PROPERTY PUBLIC Value : ETcVnKeypointDetectionTypeFAST
GET
Value := activeData;
END_GET
SET
activeData := Value;
END_SET
END_PROPERTY

END_FUNCTION_BLOCK

// Datatypes/Enums/_ETcVnLineType
{attribute 'linkalways'} 
{attribute 'no_explicit_call' := 'This FB is a CLASS and must be accessed using methods or properties'}
{attribute 'enable_dynamic_creation'}
FUNCTION_BLOCK _ETcVnLineType EXTENDS EnumDatatypeBase
VAR
	localData : ETcVnLineType;
	activeData : REFERENCE TO ETcVnLineType;
	enumBaseDatatype : _DINT(localData);
END_VAR

METHOD PROTECTED SetBaseDatatypeReference
VAR_INPUT
END_VAR
enumBaseDatatype.MakeReferenceTo(activeData);
END_METHOD

PROPERTY PUBLIC Address : PVOID
GET
Address := ADR(activeData);
END_GET
END_PROPERTY

METHOD PUBLIC ClearReference
VAR_INPUT
END_VAR
activeData REF= localData;
SetBaseDatatypeReference();
END_METHOD

PROPERTY PUBLIC Size : UDINT
GET
Size := SIZEOF(activeData);
END_GET
END_PROPERTY

METHOD FB_init : BOOL
VAR_INPUT
	bInitRetains : BOOL; // if TRUE, the retain variables are initialized (warm start / cold start)
	bInCopyCode : BOOL;  // if TRUE, the instance afterwards gets moved into the copy code (online change)
	InitialValue : ETcVnLineType;
END_VAR
localData := InitialValue;
AddBaseDatatype(enumBaseDatatype);
ClearReference();

AddLocalEnumeration('TCVN_LT_4_CONNECTED', ETcVnLineType.TCVN_LT_4_CONNECTED);
AddLocalEnumeration('TCVN_LT_8_CONNECTED', ETcVnLineType.TCVN_LT_8_CONNECTED);
AddLocalEnumeration('TCVN_LT_ANTIALIASED', ETcVnLineType.TCVN_LT_ANTIALIASED);
END_METHOD

METHOD PRIVATE AddLocalEnumeration
VAR_INPUT
	Enumeration : T_MAXSTRING;
	Value : ETcVnLineType;
END_VAR
AddEnumeration(Enumeration, Value);
END_METHOD

METHOD IsEnumeratorValueEqual : BOOL
VAR_INPUT
	Enumerator : I_KeyValueForwardEnumerator;
END_VAR
VAR
	storedValue : ETcVnLineType;
END_VAR
IF NOT Enumerator.TryGet(storedValue) THEN
	RETURN;
END_IF

IsEnumeratorValueEqual := storedValue = activeData;
END_METHOD

METHOD PUBLIC Clone : I_Datatype
VAR
    pClone : POINTER TO _ETcVnLineType;
END_VAR
pClone := __NEW(_ETcVnLineType(InitialValue := Value));
Clone := pClone^;
END_METHOD

PROPERTY PUBLIC Identifier : T_MAXSTRING
GET
Identifier := 'ETcVnLineType';
END_GET
END_PROPERTY

METHOD PUBLIC MakeReferenceTo
VAR_INPUT
	ReferenceTarget : REFERENCE TO ETcVnLineType;
END_VAR
activeData REF= ReferenceTarget;
SetBaseDatatypeReference();
END_METHOD

METHOD TryMakeReferenceTo : BOOL
VAR_INPUT
	Target : I_Datatype;
END_VAR
VAR
	pTargetData : POINTER TO ETcVnLineType;
END_VAR
IF NOT IsEquivalentTo(Target) THEN
	RETURN;
END_IF

pTargetData := Target.Address;
activeData REF= pTargetData^;
SetBaseDatatypeReference();
TryMakeReferenceTo := TRUE;
END_METHOD

PROPERTY PUBLIC Value : ETcVnLineType
GET
Value := activeData;
END_GET
SET
activeData := Value;
END_SET
END_PROPERTY

END_FUNCTION_BLOCK

// Datatypes/Enums/_ETcVnMorphologicalOperator
{attribute 'linkalways'} 
{attribute 'no_explicit_call' := 'This FB is a CLASS and must be accessed using methods or properties'}
{attribute 'enable_dynamic_creation'}
FUNCTION_BLOCK _ETcVnMorphologicalOperator EXTENDS EnumDatatypeBase
VAR
	localData : ETcVnMorphologicalOperator;
	activeData : REFERENCE TO ETcVnMorphologicalOperator;
	enumBaseDatatype : _DINT(localData);
END_VAR

METHOD PROTECTED SetBaseDatatypeReference
VAR_INPUT
END_VAR
enumBaseDatatype.MakeReferenceTo(activeData);
END_METHOD

PROPERTY PUBLIC Address : PVOID
GET
Address := ADR(activeData);
END_GET
END_PROPERTY

METHOD PUBLIC ClearReference
VAR_INPUT
END_VAR
activeData REF= localData;
SetBaseDatatypeReference();
END_METHOD

PROPERTY PUBLIC Size : UDINT
GET
Size := SIZEOF(activeData);
END_GET
END_PROPERTY

METHOD FB_init : BOOL
VAR_INPUT
	bInitRetains : BOOL; // if TRUE, the retain variables are initialized (warm start / cold start)
	bInCopyCode : BOOL;  // if TRUE, the instance afterwards gets moved into the copy code (online change)
	InitialValue : ETcVnMorphologicalOperator;
END_VAR
localData := InitialValue;
AddBaseDatatype(enumBaseDatatype);
ClearReference();

AddLocalEnumeration('TCVN_MO_EROSION', ETcVnMorphologicalOperator.TCVN_MO_EROSION);
AddLocalEnumeration('TCVN_MO_DILATION', ETcVnMorphologicalOperator.TCVN_MO_DILATION);
AddLocalEnumeration('TCVN_MO_OPENING', ETcVnMorphologicalOperator.TCVN_MO_OPENING);
AddLocalEnumeration('TCVN_MO_CLOSING', ETcVnMorphologicalOperator.TCVN_MO_CLOSING);
AddLocalEnumeration('TCVN_MO_GRADIENT', ETcVnMorphologicalOperator.TCVN_MO_GRADIENT);
AddLocalEnumeration('TCVN_MO_WHITE_TOPHAT', .TCVN_MO_WHITE_TOPHAT);
AddLocalEnumeration('TCVN_MO_BLACK_TOPHAT', ETcVnMorphologicalOperator.TCVN_MO_BLACK_TOPHAT);
AddLocalEnumeration('TCVN_MO_OPENING_BY_RECONSTRUCTION', ETcVnMorphologicalOperator.TCVN_MO_OPENING_BY_RECONSTRUCTION);
AddLocalEnumeration('TCVN_MO_CLOSING_BY_RECONSTRUCTION', ETcVnMorphologicalOperator.TCVN_MO_CLOSING_BY_RECONSTRUCTION);
AddLocalEnumeration('TCVN_MO_WHITE_TOPHAT_BY_RECONSTRUCTION', ETcVnMorphologicalOperator.TCVN_MO_WHITE_TOPHAT_BY_RECONSTRUCTION);
AddLocalEnumeration('TCVN_MO_BLACK_TOPHAT_BY_RECONSTRUCTION', ETcVnMorphologicalOperator.TCVN_MO_BLACK_TOPHAT_BY_RECONSTRUCTION);
END_METHOD

METHOD PRIVATE AddLocalEnumeration
VAR_INPUT
	Enumeration : T_MAXSTRING;
	Value : ETcVnMorphologicalOperator;
END_VAR
AddEnumeration(Enumeration, Value);
END_METHOD

METHOD IsEnumeratorValueEqual : BOOL
VAR_INPUT
	Enumerator : I_KeyValueForwardEnumerator;
END_VAR
VAR
	storedValue : ETcVnMorphologicalOperator;
END_VAR
IF NOT Enumerator.TryGet(storedValue) THEN
	RETURN;
END_IF

IsEnumeratorValueEqual := storedValue = activeData;
END_METHOD

METHOD PUBLIC Clone : I_Datatype
VAR
    pClone : POINTER TO _ETcVnMorphologicalOperator;
END_VAR
pClone := __NEW(_ETcVnMorphologicalOperator(InitialValue := Value));
Clone := pClone^;
END_METHOD

PROPERTY PUBLIC Identifier : T_MAXSTRING
GET
Identifier := 'ETcVnMorphologicalOperator';
END_GET
END_PROPERTY

METHOD PUBLIC MakeReferenceTo
VAR_INPUT
	ReferenceTarget : REFERENCE TO ETcVnMorphologicalOperator;
END_VAR
activeData REF= ReferenceTarget;
SetBaseDatatypeReference();
END_METHOD

METHOD TryMakeReferenceTo : BOOL
VAR_INPUT
	Target : I_Datatype;
END_VAR
VAR
	pTargetData : POINTER TO ETcVnMorphologicalOperator;
END_VAR
IF NOT IsEquivalentTo(Target) THEN
	RETURN;
END_IF

pTargetData := Target.Address;
activeData REF= pTargetData^;
SetBaseDatatypeReference();
TryMakeReferenceTo := TRUE;
END_METHOD

PROPERTY PUBLIC Value : ETcVnMorphologicalOperator
GET
Value := activeData;
END_GET
SET
activeData := Value;
END_SET
END_PROPERTY

END_FUNCTION_BLOCK

// Datatypes/Enums/_ETcVnNormalizationType
{attribute 'linkalways'} 
{attribute 'no_explicit_call' := 'This FB is a CLASS and must be accessed using methods or properties'}
{attribute 'enable_dynamic_creation'}
FUNCTION_BLOCK _ETcVnNormalizationType EXTENDS EnumDatatypeBase
VAR
	localData : ETcVnNormalizationType;
	activeData : REFERENCE TO ETcVnNormalizationType;
	enumBaseDatatype : _DINT(localData);
END_VAR

METHOD PROTECTED SetBaseDatatypeReference
VAR_INPUT
END_VAR
enumBaseDatatype.MakeReferenceTo(activeData);
END_METHOD

PROPERTY PUBLIC Address : PVOID
GET
Address := ADR(activeData);
END_GET
END_PROPERTY

METHOD PUBLIC ClearReference
VAR_INPUT
END_VAR
activeData REF= localData;
SetBaseDatatypeReference();
END_METHOD

PROPERTY PUBLIC Size : UDINT
GET
Size := SIZEOF(activeData);
END_GET
END_PROPERTY

METHOD FB_init : BOOL
VAR_INPUT
	bInitRetains : BOOL; // if TRUE, the retain variables are initialized (warm start / cold start)
	bInCopyCode : BOOL;  // if TRUE, the instance afterwards gets moved into the copy code (online change)
	InitialValue : ETcVnNormalizationType;
END_VAR
localData := InitialValue;
AddBaseDatatype(enumBaseDatatype);
ClearReference();

AddLocalEnumeration('TCVN_NT_INF', ETcVnNormalizationType.TCVN_NT_INF);
AddLocalEnumeration('TCVN_NT_L1', ETcVnNormalizationType.TCVN_NT_L1);
AddLocalEnumeration('TCVN_NT_L2', ETcVnNormalizationType.TCVN_NT_L2);
AddLocalEnumeration('TCVN_NT_L2SQR', ETcVnNormalizationType.TCVN_NT_L2SQR);
AddLocalEnumeration('TCVN_NT_HAMMING', ETcVnNormalizationType.TCVN_NT_HAMMING);
AddLocalEnumeration('TCVN_NT_HAMMING2', ETcVnNormalizationType.TCVN_NT_HAMMING2);
AddLocalEnumeration('TCVN_NT_RELATIVE_INF', ETcVnNormalizationType.TCVN_NT_RELATIVE_INF);
AddLocalEnumeration('TCVN_NT_RELATIVE_L1', ETcVnNormalizationType.TCVN_NT_RELATIVE_L1);
AddLocalEnumeration('TCVN_NT_RELATIVE_L2', ETcVnNormalizationType.TCVN_NT_RELATIVE_L2);
AddLocalEnumeration('TCVN_NT_RELATIVE_L2SQR', ETcVnNormalizationType.TCVN_NT_RELATIVE_L2SQR);
AddLocalEnumeration('TCVN_NT_RELATIVE_HAMMING', ETcVnNormalizationType.TCVN_NT_RELATIVE_HAMMING);
AddLocalEnumeration('TCVN_NT_RELATIVE_HAMMING2', ETcVnNormalizationType.TCVN_NT_RELATIVE_HAMMING2);
AddLocalEnumeration('TCVN_NT_MINMAX', ETcVnNormalizationType.TCVN_NT_MINMAX);
END_METHOD

METHOD PRIVATE AddLocalEnumeration
VAR_INPUT
	Enumeration : T_MAXSTRING;
	Value : ETcVnNormalizationType;
END_VAR
AddEnumeration(Enumeration, Value);
END_METHOD

METHOD IsEnumeratorValueEqual : BOOL
VAR_INPUT
	Enumerator : I_KeyValueForwardEnumerator;
END_VAR
VAR
	storedValue : ETcVnNormalizationType;
END_VAR
IF NOT Enumerator.TryGet(storedValue) THEN
	RETURN;
END_IF

IsEnumeratorValueEqual := storedValue = activeData;
END_METHOD

METHOD PUBLIC Clone : I_Datatype
VAR
    pClone : POINTER TO _ETcVnNormalizationType;
END_VAR
pClone := __NEW(_ETcVnNormalizationType(InitialValue := Value));
Clone := pClone^;
END_METHOD

PROPERTY PUBLIC Identifier : T_MAXSTRING
GET
Identifier := 'ETcVnNormalizationType';
END_GET
END_PROPERTY

METHOD PUBLIC MakeReferenceTo
VAR_INPUT
	ReferenceTarget : REFERENCE TO ETcVnNormalizationType;
END_VAR
activeData REF= ReferenceTarget;
SetBaseDatatypeReference();
END_METHOD

METHOD TryMakeReferenceTo : BOOL
VAR_INPUT
	Target : I_Datatype;
END_VAR
VAR
	pTargetData : POINTER TO ETcVnNormalizationType;
END_VAR
IF NOT IsEquivalentTo(Target) THEN
	RETURN;
END_IF

pTargetData := Target.Address;
activeData REF= pTargetData^;
SetBaseDatatypeReference();
TryMakeReferenceTo := TRUE;
END_METHOD

PROPERTY PUBLIC Value : ETcVnNormalizationType
GET
Value := activeData;
END_GET
SET
activeData := Value;
END_SET
END_PROPERTY

END_FUNCTION_BLOCK

// Datatypes/Enums/_ETcVnOrientationMethod
{attribute 'linkalways'} 
{attribute 'no_explicit_call' := 'This FB is a CLASS and must be accessed using methods or properties'}
{attribute 'enable_dynamic_creation'}
FUNCTION_BLOCK _ETcVnOrientationMethod EXTENDS EnumDatatypeBase
VAR
	localData : ETcVnOrientationMethod;
	activeData : REFERENCE TO ETcVnOrientationMethod;
	enumBaseDatatype : _DINT(localData);
END_VAR

METHOD PROTECTED SetBaseDatatypeReference
VAR_INPUT
END_VAR
enumBaseDatatype.MakeReferenceTo(activeData);
END_METHOD

PROPERTY PUBLIC Address : PVOID
GET
Address := ADR(activeData);
END_GET
END_PROPERTY

METHOD PUBLIC ClearReference
VAR_INPUT
END_VAR
activeData REF= localData;
SetBaseDatatypeReference();
END_METHOD

PROPERTY PUBLIC Size : UDINT
GET
Size := SIZEOF(activeData);
END_GET
END_PROPERTY

METHOD FB_init : BOOL
VAR_INPUT
	bInitRetains : BOOL; // if TRUE, the retain variables are initialized (warm start / cold start)
	bInCopyCode : BOOL;  // if TRUE, the instance afterwards gets moved into the copy code (online change)
	InitialValue : ETcVnOrientationMethod;
END_VAR
localData := InitialValue;
AddBaseDatatype(enumBaseDatatype);
ClearReference();

AddLocalEnumeration('TCVN_OM_PCA', ETcVnOrientationMethod.TCVN_OM_PCA);
AddLocalEnumeration('TCVN_OM_FITELLIPSE', ETcVnOrientationMethod.TCVN_OM_FITELLIPSE);
AddLocalEnumeration('TCVN_OM_MOMENTS', ETcVnOrientationMethod.TCVN_OM_MOMENTS);
AddLocalEnumeration('TCVN_OM_ENCLOSINGRECT', ETcVnOrientationMethod.TCVN_OM_ENCLOSINGRECT);
END_METHOD

METHOD PRIVATE AddLocalEnumeration
VAR_INPUT
	Enumeration : T_MAXSTRING;
	Value : ETcVnOrientationMethod;
END_VAR
AddEnumeration(Enumeration, Value);
END_METHOD

METHOD IsEnumeratorValueEqual : BOOL
VAR_INPUT
	Enumerator : I_KeyValueForwardEnumerator;
END_VAR
VAR
	storedValue : ETcVnOrientationMethod;
END_VAR
IF NOT Enumerator.TryGet(storedValue) THEN
	RETURN;
END_IF

IsEnumeratorValueEqual := storedValue = activeData;
END_METHOD

METHOD PUBLIC Clone : I_Datatype
VAR
    pClone : POINTER TO _ETcVnOrientationMethod;
END_VAR
pClone := __NEW(_ETcVnOrientationMethod(InitialValue := Value));
Clone := pClone^;
END_METHOD

PROPERTY PUBLIC Identifier : T_MAXSTRING
GET
Identifier := 'ETcVnOrientationMethod';
END_GET
END_PROPERTY

METHOD PUBLIC MakeReferenceTo
VAR_INPUT
	ReferenceTarget : REFERENCE TO ETcVnOrientationMethod;
END_VAR
activeData REF= ReferenceTarget;
SetBaseDatatypeReference();
END_METHOD

METHOD TryMakeReferenceTo : BOOL
VAR_INPUT
	Target : I_Datatype;
END_VAR
VAR
	pTargetData : POINTER TO ETcVnOrientationMethod;
END_VAR
IF NOT IsEquivalentTo(Target) THEN
	RETURN;
END_IF

pTargetData := Target.Address;
activeData REF= pTargetData^;
SetBaseDatatypeReference();
TryMakeReferenceTo := TRUE;
END_METHOD

PROPERTY PUBLIC Value : ETcVnOrientationMethod
GET
Value := activeData;
END_GET
SET
activeData := Value;
END_SET
END_PROPERTY

END_FUNCTION_BLOCK

// Datatypes/Enums/_ETcVnPixelConnectivity
{attribute 'linkalways'} 
{attribute 'no_explicit_call' := 'This FB is a CLASS and must be accessed using methods or properties'}
{attribute 'enable_dynamic_creation'}
FUNCTION_BLOCK _ETcVnPixelConnectivity EXTENDS EnumDatatypeBase
VAR
	localData : ETcVnPixelConnectivity;
	activeData : REFERENCE TO ETcVnPixelConnectivity;
	enumBaseDatatype : _DINT(localData);
END_VAR

METHOD PROTECTED SetBaseDatatypeReference
VAR_INPUT
END_VAR
enumBaseDatatype.MakeReferenceTo(activeData);
END_METHOD

PROPERTY PUBLIC Address : PVOID
GET
Address := ADR(activeData);
END_GET
END_PROPERTY

METHOD PUBLIC ClearReference
VAR_INPUT
END_VAR
activeData REF= localData;
SetBaseDatatypeReference();
END_METHOD

PROPERTY PUBLIC Size : UDINT
GET
Size := SIZEOF(activeData);
END_GET
END_PROPERTY

METHOD FB_init : BOOL
VAR_INPUT
	bInitRetains : BOOL; // if TRUE, the retain variables are initialized (warm start / cold start)
	bInCopyCode : BOOL;  // if TRUE, the instance afterwards gets moved into the copy code (online change)
	InitialValue : ETcVnPixelConnectivity;
END_VAR
localData := InitialValue;
AddBaseDatatype(enumBaseDatatype);
ClearReference();

AddLocalEnumeration('TCVN_PC_4', ETcVnPixelConnectivity.TCVN_PC_4);
AddLocalEnumeration('TCVN_PC_8', ETcVnPixelConnectivity.TCVN_PC_8);
END_METHOD

METHOD PRIVATE AddLocalEnumeration
VAR_INPUT
	Enumeration : T_MAXSTRING;
	Value : ETcVnPixelConnectivity;
END_VAR
AddEnumeration(Enumeration, Value);
END_METHOD

METHOD IsEnumeratorValueEqual : BOOL
VAR_INPUT
	Enumerator : I_KeyValueForwardEnumerator;
END_VAR
VAR
	storedValue : ETcVnPixelConnectivity;
END_VAR
IF NOT Enumerator.TryGet(storedValue) THEN
	RETURN;
END_IF

IsEnumeratorValueEqual := storedValue = activeData;
END_METHOD

METHOD PUBLIC Clone : I_Datatype
VAR
    pClone : POINTER TO _ETcVnPixelConnectivity;
END_VAR
pClone := __NEW(_ETcVnPixelConnectivity(InitialValue := Value));
Clone := pClone^;
END_METHOD

PROPERTY PUBLIC Identifier : T_MAXSTRING
GET
Identifier := 'ETcVnPixelConnectivity';
END_GET
END_PROPERTY

METHOD PUBLIC MakeReferenceTo
VAR_INPUT
	ReferenceTarget : REFERENCE TO ETcVnPixelConnectivity;
END_VAR
activeData REF= ReferenceTarget;
SetBaseDatatypeReference();
END_METHOD

METHOD TryMakeReferenceTo : BOOL
VAR_INPUT
	Target : I_Datatype;
END_VAR
VAR
	pTargetData : POINTER TO ETcVnPixelConnectivity;
END_VAR
IF NOT IsEquivalentTo(Target) THEN
	RETURN;
END_IF

pTargetData := Target.Address;
activeData REF= pTargetData^;
SetBaseDatatypeReference();
TryMakeReferenceTo := TRUE;
END_METHOD

PROPERTY PUBLIC Value : ETcVnPixelConnectivity
GET
Value := activeData;
END_GET
SET
activeData := Value;
END_SET
END_PROPERTY

END_FUNCTION_BLOCK

// Datatypes/Enums/_ETcVnRectangleIntersection
{attribute 'linkalways'} 
{attribute 'no_explicit_call' := 'This FB is a CLASS and must be accessed using methods or properties'}
{attribute 'enable_dynamic_creation'}
FUNCTION_BLOCK _ETcVnRectangleIntersection EXTENDS EnumDatatypeBase
VAR
	localData : ETcVnRectangleIntersection;
	activeData : REFERENCE TO ETcVnRectangleIntersection;
	enumBaseDatatype : _DINT(localData);
END_VAR

METHOD PROTECTED SetBaseDatatypeReference
VAR_INPUT
END_VAR
enumBaseDatatype.MakeReferenceTo(activeData);
END_METHOD

PROPERTY PUBLIC Address : PVOID
GET
Address := ADR(activeData);
END_GET
END_PROPERTY

METHOD PUBLIC ClearReference
VAR_INPUT
END_VAR
activeData REF= localData;
SetBaseDatatypeReference();
END_METHOD

PROPERTY PUBLIC Size : UDINT
GET
Size := SIZEOF(activeData);
END_GET
END_PROPERTY

METHOD FB_init : BOOL
VAR_INPUT
	bInitRetains : BOOL; // if TRUE, the retain variables are initialized (warm start / cold start)
	bInCopyCode : BOOL;  // if TRUE, the instance afterwards gets moved into the copy code (online change)
	InitialValue : ETcVnRectangleIntersection;
END_VAR
localData := InitialValue;
AddBaseDatatype(enumBaseDatatype);
ClearReference();

AddLocalEnumeration('TCVN_RI_NONE', ETcVnRectangleIntersection.TCVN_RI_NONE);
AddLocalEnumeration('TCVN_RI_PARTIAL', ETcVnRectangleIntersection.TCVN_RI_PARTIAL);
AddLocalEnumeration('TCVN_RI_FULL', ETcVnRectangleIntersection.TCVN_RI_FULL);
END_METHOD

METHOD PRIVATE AddLocalEnumeration
VAR_INPUT
	Enumeration : T_MAXSTRING;
	Value : ETcVnRectangleIntersection;
END_VAR
AddEnumeration(Enumeration, Value);
END_METHOD

METHOD IsEnumeratorValueEqual : BOOL
VAR_INPUT
	Enumerator : I_KeyValueForwardEnumerator;
END_VAR
VAR
	storedValue : ETcVnRectangleIntersection;
END_VAR
IF NOT Enumerator.TryGet(storedValue) THEN
	RETURN;
END_IF

IsEnumeratorValueEqual := storedValue = activeData;
END_METHOD

METHOD PUBLIC Clone : I_Datatype
VAR
    pClone : POINTER TO _ETcVnRectangleIntersection;
END_VAR
pClone := __NEW(_ETcVnRectangleIntersection(InitialValue := Value));
Clone := pClone^;
END_METHOD

PROPERTY PUBLIC Identifier : T_MAXSTRING
GET
Identifier := 'ETcVnRectangleIntersection';
END_GET
END_PROPERTY

METHOD PUBLIC MakeReferenceTo
VAR_INPUT
	ReferenceTarget : REFERENCE TO ETcVnRectangleIntersection;
END_VAR
activeData REF= ReferenceTarget;
SetBaseDatatypeReference();
END_METHOD

METHOD TryMakeReferenceTo : BOOL
VAR_INPUT
	Target : I_Datatype;
END_VAR
VAR
	pTargetData : POINTER TO ETcVnRectangleIntersection;
END_VAR
IF NOT IsEquivalentTo(Target) THEN
	RETURN;
END_IF

pTargetData := Target.Address;
activeData REF= pTargetData^;
SetBaseDatatypeReference();
TryMakeReferenceTo := TRUE;
END_METHOD

PROPERTY PUBLIC Value : ETcVnRectangleIntersection
GET
Value := activeData;
END_GET
SET
activeData := Value;
END_SET
END_PROPERTY

END_FUNCTION_BLOCK

// Datatypes/Enums/_ETcVnRotationAngle
{attribute 'linkalways'} 
{attribute 'no_explicit_call' := 'This FB is a CLASS and must be accessed using methods or properties'}
{attribute 'enable_dynamic_creation'}
FUNCTION_BLOCK _ETcVnRotationAngle EXTENDS EnumDatatypeBase
VAR
	localData : ETcVnRotationAngle;
	activeData : REFERENCE TO ETcVnRotationAngle;
	enumBaseDatatype : _DINT(localData);
END_VAR

METHOD PROTECTED SetBaseDatatypeReference
VAR_INPUT
END_VAR
enumBaseDatatype.MakeReferenceTo(activeData);
END_METHOD

PROPERTY PUBLIC Address : PVOID
GET
Address := ADR(activeData);
END_GET
END_PROPERTY

METHOD PUBLIC ClearReference
VAR_INPUT
END_VAR
activeData REF= localData;
SetBaseDatatypeReference();
END_METHOD

PROPERTY PUBLIC Size : UDINT
GET
Size := SIZEOF(activeData);
END_GET
END_PROPERTY

METHOD FB_init : BOOL
VAR_INPUT
	bInitRetains : BOOL; // if TRUE, the retain variables are initialized (warm start / cold start)
	bInCopyCode : BOOL;  // if TRUE, the instance afterwards gets moved into the copy code (online change)
	InitialValue : ETcVnRotationAngle;
END_VAR
localData := InitialValue;
AddBaseDatatype(enumBaseDatatype);
ClearReference();

AddLocalEnumeration('TCVN_RA_90_DEG', ETcVnRotationAngle.TCVN_RA_90_DEG);
AddLocalEnumeration('TCVN_RA_180_DEG', ETcVnRotationAngle.TCVN_RA_180_DEG);
AddLocalEnumeration('TCVN_RA_270_DEG', ETcVnRotationAngle.TCVN_RA_270_DEG);
END_METHOD

METHOD PRIVATE AddLocalEnumeration
VAR_INPUT
	Enumeration : T_MAXSTRING;
	Value : ETcVnRotationAngle;
END_VAR
AddEnumeration(Enumeration, Value);
END_METHOD

METHOD IsEnumeratorValueEqual : BOOL
VAR_INPUT
	Enumerator : I_KeyValueForwardEnumerator;
END_VAR
VAR
	storedValue : ETcVnRotationAngle;
END_VAR
IF NOT Enumerator.TryGet(storedValue) THEN
	RETURN;
END_IF

IsEnumeratorValueEqual := storedValue = activeData;
END_METHOD

METHOD PUBLIC Clone : I_Datatype
VAR
    pClone : POINTER TO _ETcVnRotationAngle;
END_VAR
pClone := __NEW(_ETcVnRotationAngle(InitialValue := Value));
Clone := pClone^;
END_METHOD

PROPERTY PUBLIC Identifier : T_MAXSTRING
GET
Identifier := 'ETcVnRotationAngle';
END_GET
END_PROPERTY

METHOD PUBLIC MakeReferenceTo
VAR_INPUT
	ReferenceTarget : REFERENCE TO ETcVnRotationAngle;
END_VAR
activeData REF= ReferenceTarget;
SetBaseDatatypeReference();
END_METHOD

METHOD TryMakeReferenceTo : BOOL
VAR_INPUT
	Target : I_Datatype;
END_VAR
VAR
	pTargetData : POINTER TO ETcVnRotationAngle;
END_VAR
IF NOT IsEquivalentTo(Target) THEN
	RETURN;
END_IF

pTargetData := Target.Address;
activeData REF= pTargetData^;
SetBaseDatatypeReference();
TryMakeReferenceTo := TRUE;
END_METHOD

PROPERTY PUBLIC Value : ETcVnRotationAngle
GET
Value := activeData;
END_GET
SET
activeData := Value;
END_SET
END_PROPERTY

END_FUNCTION_BLOCK

// Datatypes/Enums/_ETcVnSignedNormalization
{attribute 'linkalways'} 
{attribute 'no_explicit_call' := 'This FB is a CLASS and must be accessed using methods or properties'}
{attribute 'enable_dynamic_creation'}
FUNCTION_BLOCK _ETcVnSignedNormalization EXTENDS EnumDatatypeBase
VAR
	localData : ETcVnSignedNormalization;
	activeData : REFERENCE TO ETcVnSignedNormalization;
	enumBaseDatatype : _INT(localData);
END_VAR

METHOD PROTECTED SetBaseDatatypeReference
VAR_INPUT
END_VAR
enumBaseDatatype.MakeReferenceTo(activeData);
END_METHOD

PROPERTY PUBLIC Address : PVOID
GET
Address := ADR(activeData);
END_GET
END_PROPERTY

METHOD PUBLIC ClearReference
VAR_INPUT
END_VAR
activeData REF= localData;
SetBaseDatatypeReference();
END_METHOD

PROPERTY PUBLIC Size : UDINT
GET
Size := SIZEOF(activeData);
END_GET
END_PROPERTY

METHOD FB_init : BOOL
VAR_INPUT
	bInitRetains : BOOL; // if TRUE, the retain variables are initialized (warm start / cold start)
	bInCopyCode : BOOL;  // if TRUE, the instance afterwards gets moved into the copy code (online change)
	InitialValue : ETcVnSignedNormalization;
END_VAR
localData := InitialValue;
AddBaseDatatype(enumBaseDatatype);
ClearReference();

AddLocalEnumeration('TCVN_SN_FIX_ZERO', ETcVnSignedNormalization.TCVN_SN_FIX_ZERO);
AddLocalEnumeration('TCVN_SN_FULL_SCALE', ETcVnSignedNormalization.TCVN_SN_FULL_SCALE);
END_METHOD

METHOD PRIVATE AddLocalEnumeration
VAR_INPUT
	Enumeration : T_MAXSTRING;
	Value : ETcVnSignedNormalization;
END_VAR
AddEnumeration(Enumeration, Value);
END_METHOD

METHOD IsEnumeratorValueEqual : BOOL
VAR_INPUT
	Enumerator : I_KeyValueForwardEnumerator;
END_VAR
VAR
	storedValue : ETcVnSignedNormalization;
END_VAR
IF NOT Enumerator.TryGet(storedValue) THEN
	RETURN;
END_IF

IsEnumeratorValueEqual := storedValue = activeData;
END_METHOD

METHOD PUBLIC Clone : I_Datatype
VAR
    pClone : POINTER TO _ETcVnSignedNormalization;
END_VAR
pClone := __NEW(_ETcVnSignedNormalization(InitialValue := Value));
Clone := pClone^;
END_METHOD

PROPERTY PUBLIC Identifier : T_MAXSTRING
GET
Identifier := 'ETcVnSignedNormalization';
END_GET
END_PROPERTY

METHOD PUBLIC MakeReferenceTo
VAR_INPUT
	ReferenceTarget : REFERENCE TO ETcVnSignedNormalization;
END_VAR
activeData REF= ReferenceTarget;
SetBaseDatatypeReference();
END_METHOD

METHOD TryMakeReferenceTo : BOOL
VAR_INPUT
	Target : I_Datatype;
END_VAR
VAR
	pTargetData : POINTER TO ETcVnSignedNormalization;
END_VAR
IF NOT IsEquivalentTo(Target) THEN
	RETURN;
END_IF

pTargetData := Target.Address;
activeData REF= pTargetData^;
SetBaseDatatypeReference();
TryMakeReferenceTo := TRUE;
END_METHOD

PROPERTY PUBLIC Value : ETcVnSignedNormalization
GET
Value := activeData;
END_GET
SET
activeData := Value;
END_SET
END_PROPERTY

END_FUNCTION_BLOCK

// Datatypes/Enums/_ETcVnStructuringElementShape
{attribute 'linkalways'} 
{attribute 'no_explicit_call' := 'This FB is a CLASS and must be accessed using methods or properties'}
{attribute 'enable_dynamic_creation'}
FUNCTION_BLOCK _ETcVnStructuringElementShape EXTENDS EnumDatatypeBase
VAR
	localData : ETcVnStructuringElementShape;
	activeData : REFERENCE TO ETcVnStructuringElementShape;
	enumBaseDatatype : _DINT(localData);
END_VAR

METHOD PROTECTED SetBaseDatatypeReference
VAR_INPUT
END_VAR
enumBaseDatatype.MakeReferenceTo(activeData);
END_METHOD

PROPERTY PUBLIC Address : PVOID
GET
Address := ADR(activeData);
END_GET
END_PROPERTY

METHOD PUBLIC ClearReference
VAR_INPUT
END_VAR
activeData REF= localData;
SetBaseDatatypeReference();
END_METHOD

PROPERTY PUBLIC Size : UDINT
GET
Size := SIZEOF(activeData);
END_GET
END_PROPERTY

METHOD FB_init : BOOL
VAR_INPUT
	bInitRetains : BOOL; // if TRUE, the retain variables are initialized (warm start / cold start)
	bInCopyCode : BOOL;  // if TRUE, the instance afterwards gets moved into the copy code (online change)
	InitialValue : ETcVnStructuringElementShape;
END_VAR
localData := InitialValue;
AddBaseDatatype(enumBaseDatatype);
ClearReference();

AddLocalEnumeration('TCVN_SES_RECTANGLE', ETcVnStructuringElementShape.TCVN_SES_RECTANGLE);
AddLocalEnumeration('TCVN_SES_CROSS', ETcVnStructuringElementShape.TCVN_SES_CROSS);
AddLocalEnumeration('TCVN_SES_ELLIPSE', ETcVnStructuringElementShape.TCVN_SES_ELLIPSE);
END_METHOD

METHOD PRIVATE AddLocalEnumeration
VAR_INPUT
	Enumeration : T_MAXSTRING;
	Value : ETcVnStructuringElementShape;
END_VAR
AddEnumeration(Enumeration, Value);
END_METHOD

METHOD IsEnumeratorValueEqual : BOOL
VAR_INPUT
	Enumerator : I_KeyValueForwardEnumerator;
END_VAR
VAR
	storedValue : ETcVnStructuringElementShape;
END_VAR
IF NOT Enumerator.TryGet(storedValue) THEN
	RETURN;
END_IF

IsEnumeratorValueEqual := storedValue = activeData;
END_METHOD

METHOD PUBLIC Clone : I_Datatype
VAR
    pClone : POINTER TO _ETcVnStructuringElementShape;
END_VAR
pClone := __NEW(_ETcVnStructuringElementShape(InitialValue := Value));
Clone := pClone^;
END_METHOD

PROPERTY PUBLIC Identifier : T_MAXSTRING
GET
Identifier := 'ETcVnStructuringElementShape';
END_GET
END_PROPERTY

METHOD PUBLIC MakeReferenceTo
VAR_INPUT
	ReferenceTarget : REFERENCE TO ETcVnStructuringElementShape;
END_VAR
activeData REF= ReferenceTarget;
SetBaseDatatypeReference();
END_METHOD

METHOD TryMakeReferenceTo : BOOL
VAR_INPUT
	Target : I_Datatype;
END_VAR
VAR
	pTargetData : POINTER TO ETcVnStructuringElementShape;
END_VAR
IF NOT IsEquivalentTo(Target) THEN
	RETURN;
END_IF

pTargetData := Target.Address;
activeData REF= pTargetData^;
SetBaseDatatypeReference();
TryMakeReferenceTo := TRUE;
END_METHOD

PROPERTY PUBLIC Value : ETcVnStructuringElementShape
GET
Value := activeData;
END_GET
SET
activeData := Value;
END_SET
END_PROPERTY

END_FUNCTION_BLOCK

// Datatypes/Enums/_ETcVnTemplateMatchMethod
{attribute 'linkalways'} 
{attribute 'no_explicit_call' := 'This FB is a CLASS and must be accessed using methods or properties'}
{attribute 'enable_dynamic_creation'}
FUNCTION_BLOCK _ETcVnTemplateMatchMethod EXTENDS EnumDatatypeBase
VAR
	localData : ETcVnTemplateMatchMethod;
	activeData : REFERENCE TO ETcVnTemplateMatchMethod;
	enumBaseDatatype : _DINT(localData);
END_VAR

METHOD PROTECTED SetBaseDatatypeReference
VAR_INPUT
END_VAR
enumBaseDatatype.MakeReferenceTo(activeData);
END_METHOD

PROPERTY PUBLIC Address : PVOID
GET
Address := ADR(activeData);
END_GET
END_PROPERTY

METHOD PUBLIC ClearReference
VAR_INPUT
END_VAR
activeData REF= localData;
SetBaseDatatypeReference();
END_METHOD

PROPERTY PUBLIC Size : UDINT
GET
Size := SIZEOF(activeData);
END_GET
END_PROPERTY

METHOD FB_init : BOOL
VAR_INPUT
	bInitRetains : BOOL; // if TRUE, the retain variables are initialized (warm start / cold start)
	bInCopyCode : BOOL;  // if TRUE, the instance afterwards gets moved into the copy code (online change)
	InitialValue : ETcVnTemplateMatchMethod;
END_VAR
localData := InitialValue;
AddBaseDatatype(enumBaseDatatype);
ClearReference();

AddLocalEnumeration('TCVN_TMM_SQDIFF', ETcVnTemplateMatchMethod.TCVN_TMM_SQDIFF);
AddLocalEnumeration('TCVN_TMM_SQDIFF_NORMED', ETcVnTemplateMatchMethod.TCVN_TMM_SQDIFF_NORMED);
AddLocalEnumeration('TCVN_TMM_CCORR', ETcVnTemplateMatchMethod.TCVN_TMM_CCORR);
AddLocalEnumeration('TCVN_TMM_CCORR_NORMED', ETcVnTemplateMatchMethod.TCVN_TMM_CCORR_NORMED);
AddLocalEnumeration('TCVN_TMM_CCOEFF', ETcVnTemplateMatchMethod.TCVN_TMM_CCOEFF);
AddLocalEnumeration('TCVN_TMM_CCOEFF_NORMED', ETcVnTemplateMatchMethod.TCVN_TMM_CCOEFF_NORMED);
END_METHOD

METHOD PRIVATE AddLocalEnumeration
VAR_INPUT
	Enumeration : T_MAXSTRING;
	Value : ETcVnTemplateMatchMethod;
END_VAR
AddEnumeration(Enumeration, Value);
END_METHOD

METHOD IsEnumeratorValueEqual : BOOL
VAR_INPUT
	Enumerator : I_KeyValueForwardEnumerator;
END_VAR
VAR
	storedValue : ETcVnTemplateMatchMethod;
END_VAR
IF NOT Enumerator.TryGet(storedValue) THEN
	RETURN;
END_IF

IsEnumeratorValueEqual := storedValue = activeData;
END_METHOD

METHOD PUBLIC Clone : I_Datatype
VAR
    pClone : POINTER TO _ETcVnTemplateMatchMethod;
END_VAR
pClone := __NEW(_ETcVnTemplateMatchMethod(InitialValue := Value));
Clone := pClone^;
END_METHOD

PROPERTY PUBLIC Identifier : T_MAXSTRING
GET
Identifier := 'ETcVnTemplateMatchMethod';
END_GET
END_PROPERTY

METHOD PUBLIC MakeReferenceTo
VAR_INPUT
	ReferenceTarget : REFERENCE TO ETcVnTemplateMatchMethod;
END_VAR
activeData REF= ReferenceTarget;
SetBaseDatatypeReference();
END_METHOD

METHOD TryMakeReferenceTo : BOOL
VAR_INPUT
	Target : I_Datatype;
END_VAR
VAR
	pTargetData : POINTER TO ETcVnTemplateMatchMethod;
END_VAR
IF NOT IsEquivalentTo(Target) THEN
	RETURN;
END_IF

pTargetData := Target.Address;
activeData REF= pTargetData^;
SetBaseDatatypeReference();
TryMakeReferenceTo := TRUE;
END_METHOD

PROPERTY PUBLIC Value : ETcVnTemplateMatchMethod
GET
Value := activeData;
END_GET
SET
activeData := Value;
END_SET
END_PROPERTY

END_FUNCTION_BLOCK

// Datatypes/Enums/_ETcVnThresholdType
{attribute 'linkalways'} 
{attribute 'no_explicit_call' := 'This FB is a CLASS and must be accessed using methods or properties'}
{attribute 'enable_dynamic_creation'}
FUNCTION_BLOCK _ETcVnThresholdType EXTENDS EnumDatatypeBase
VAR
	localData : ETcVnThresholdType;
	activeData : REFERENCE TO ETcVnThresholdType;
	enumBaseDatatype : _DINT(localData);
END_VAR

METHOD PROTECTED SetBaseDatatypeReference
VAR_INPUT
END_VAR
enumBaseDatatype.MakeReferenceTo(activeData);
END_METHOD

PROPERTY PUBLIC Address : PVOID
GET
Address := ADR(activeData);
END_GET
END_PROPERTY

METHOD PUBLIC ClearReference
VAR_INPUT
END_VAR
activeData REF= localData;
SetBaseDatatypeReference();
END_METHOD

PROPERTY PUBLIC Size : UDINT
GET
Size := SIZEOF(activeData);
END_GET
END_PROPERTY

METHOD FB_init : BOOL
VAR_INPUT
	bInitRetains : BOOL; // if TRUE, the retain variables are initialized (warm start / cold start)
	bInCopyCode : BOOL;  // if TRUE, the instance afterwards gets moved into the copy code (online change)
	InitialValue : ETcVnThresholdType;
END_VAR
localData := InitialValue;
AddBaseDatatype(enumBaseDatatype);
ClearReference();

AddLocalEnumeration('TCVN_TT_BINARY', ETcVnThresholdType.TCVN_TT_BINARY);
AddLocalEnumeration('TCVN_TT_BINARY_INV', ETcVnThresholdType.TCVN_TT_BINARY_INV);
AddLocalEnumeration('TCVN_TT_TRUNC', ETcVnThresholdType.TCVN_TT_TRUNC);
AddLocalEnumeration('TCVN_TT_TOZERO', ETcVnThresholdType.TCVN_TT_TOZERO);
AddLocalEnumeration('TCVN_TT_TOZERO_INV', ETcVnThresholdType.TCVN_TT_TOZERO_INV);
AddLocalEnumeration('TCVN_TT_OTSU_BINARY', ETcVnThresholdType.TCVN_TT_OTSU_BINARY);
AddLocalEnumeration('TCVN_TT_OTSU_BINARY_INV', ETcVnThresholdType.TCVN_TT_OTSU_BINARY_INV);
AddLocalEnumeration('TCVN_TT_OTSU_TRUNC', ETcVnThresholdType.TCVN_TT_OTSU_TRUNC);
AddLocalEnumeration('TCVN_TT_OTSU_TOZERO', ETcVnThresholdType.TCVN_TT_OTSU_TOZERO);
AddLocalEnumeration('TCVN_TT_OTSU_TOZERO_INV', ETcVnThresholdType.TCVN_TT_OTSU_TOZERO_INV);
AddLocalEnumeration('TCVN_TT_TRIANGLE_BINARY', ETcVnThresholdType.TCVN_TT_TRIANGLE_BINARY);
AddLocalEnumeration('TCVN_TT_TRIANGLE_BINARY_INV', ETcVnThresholdType.TCVN_TT_TRIANGLE_BINARY_INV);
AddLocalEnumeration('TCVN_TT_TRIANGLE_TRUNC', ETcVnThresholdType.TCVN_TT_TRIANGLE_TRUNC);
AddLocalEnumeration('TCVN_TT_TRIANGLE_TOZERO', ETcVnThresholdType.TCVN_TT_TRIANGLE_TOZERO);
AddLocalEnumeration('TCVN_TT_TRIANGLE_TOZERO_INV', ETcVnThresholdType.TCVN_TT_TRIANGLE_TOZERO_INV);
END_METHOD

METHOD PRIVATE AddLocalEnumeration
VAR_INPUT
	Enumeration : T_MAXSTRING;
	Value : ETcVnThresholdType;
END_VAR
AddEnumeration(Enumeration, Value);
END_METHOD

METHOD IsEnumeratorValueEqual : BOOL
VAR_INPUT
	Enumerator : I_KeyValueForwardEnumerator;
END_VAR
VAR
	storedValue : ETcVnThresholdType;
END_VAR
IF NOT Enumerator.TryGet(storedValue) THEN
	RETURN;
END_IF

IsEnumeratorValueEqual := storedValue = activeData;
END_METHOD

METHOD PUBLIC Clone : I_Datatype
VAR
    pClone : POINTER TO _ETcVnThresholdType;
END_VAR
pClone := __NEW(_ETcVnThresholdType(InitialValue := Value));
Clone := pClone^;
END_METHOD

PROPERTY PUBLIC Identifier : T_MAXSTRING
GET
Identifier := 'ETcVnThresholdType';
END_GET
END_PROPERTY

METHOD PUBLIC MakeReferenceTo
VAR_INPUT
	ReferenceTarget : REFERENCE TO ETcVnThresholdType;
END_VAR
activeData REF= ReferenceTarget;
SetBaseDatatypeReference();
END_METHOD

METHOD TryMakeReferenceTo : BOOL
VAR_INPUT
	Target : I_Datatype;
END_VAR
VAR
	pTargetData : POINTER TO ETcVnThresholdType;
END_VAR
IF NOT IsEquivalentTo(Target) THEN
	RETURN;
END_IF

pTargetData := Target.Address;
activeData REF= pTargetData^;
SetBaseDatatypeReference();
TryMakeReferenceTo := TRUE;
END_METHOD

PROPERTY PUBLIC Value : ETcVnThresholdType
GET
Value := activeData;
END_GET
SET
activeData := Value;
END_SET
END_PROPERTY

END_FUNCTION_BLOCK

// Datatypes/Enums/_ETcVnVectorCompareMethod
{attribute 'linkalways'} 
{attribute 'no_explicit_call' := 'This FB is a CLASS and must be accessed using methods or properties'}
{attribute 'enable_dynamic_creation'}
FUNCTION_BLOCK _ETcVnVectorCompareMethod EXTENDS EnumDatatypeBase
VAR
	localData : ETcVnVectorCompareMethod;
	activeData : REFERENCE TO ETcVnVectorCompareMethod;
	enumBaseDatatype : _DINT(localData);
END_VAR

METHOD PROTECTED SetBaseDatatypeReference
VAR_INPUT
END_VAR
enumBaseDatatype.MakeReferenceTo(activeData);
END_METHOD

PROPERTY PUBLIC Address : PVOID
GET
Address := ADR(activeData);
END_GET
END_PROPERTY

METHOD PUBLIC ClearReference
VAR_INPUT
END_VAR
activeData REF= localData;
SetBaseDatatypeReference();
END_METHOD

PROPERTY PUBLIC Size : UDINT
GET
Size := SIZEOF(activeData);
END_GET
END_PROPERTY

METHOD FB_init : BOOL
VAR_INPUT
	bInitRetains : BOOL; // if TRUE, the retain variables are initialized (warm start / cold start)
	bInCopyCode : BOOL;  // if TRUE, the instance afterwards gets moved into the copy code (online change)
	InitialValue : ETcVnVectorCompareMethod;
END_VAR
localData := InitialValue;
AddBaseDatatype(enumBaseDatatype);
ClearReference();

AddLocalEnumeration('TCVN_VCM_EUCLIDEAN', ETcVnVectorCompareMethod.TCVN_VCM_EUCLIDEAN);
AddLocalEnumeration('TCVN_VCM_ELEMENTWISE', ETcVnVectorCompareMethod.TCVN_VCM_ELEMENTWISE);
END_METHOD

METHOD PRIVATE AddLocalEnumeration
VAR_INPUT
	Enumeration : T_MAXSTRING;
	Value : ETcVnVectorCompareMethod;
END_VAR
AddEnumeration(Enumeration, Value);
END_METHOD

METHOD IsEnumeratorValueEqual : BOOL
VAR_INPUT
	Enumerator : I_KeyValueForwardEnumerator;
END_VAR
VAR
	storedValue : ETcVnVectorCompareMethod;
END_VAR
IF NOT Enumerator.TryGet(storedValue) THEN
	RETURN;
END_IF

IsEnumeratorValueEqual := storedValue = activeData;
END_METHOD

METHOD PUBLIC Clone : I_Datatype
VAR
    pClone : POINTER TO _ETcVnVectorCompareMethod;
END_VAR
pClone := __NEW(_ETcVnVectorCompareMethod(InitialValue := Value));
Clone := pClone^;
END_METHOD

PROPERTY PUBLIC Identifier : T_MAXSTRING
GET
Identifier := 'ETcVnVectorCompareMethod';
END_GET
END_PROPERTY

METHOD PUBLIC MakeReferenceTo
VAR_INPUT
	ReferenceTarget : REFERENCE TO ETcVnVectorCompareMethod;
END_VAR
activeData REF= ReferenceTarget;
SetBaseDatatypeReference();
END_METHOD

METHOD TryMakeReferenceTo : BOOL
VAR_INPUT
	Target : I_Datatype;
END_VAR
VAR
	pTargetData : POINTER TO ETcVnVectorCompareMethod;
END_VAR
IF NOT IsEquivalentTo(Target) THEN
	RETURN;
END_IF

pTargetData := Target.Address;
activeData REF= pTargetData^;
SetBaseDatatypeReference();
TryMakeReferenceTo := TRUE;
END_METHOD

PROPERTY PUBLIC Value : ETcVnVectorCompareMethod
GET
Value := activeData;
END_GET
SET
activeData := Value;
END_SET
END_PROPERTY

END_FUNCTION_BLOCK

// Datatypes/Enums/_ETcVnWorldCoordinateSystem
{attribute 'linkalways'} 
{attribute 'no_explicit_call' := 'This FB is a CLASS and must be accessed using methods or properties'}
{attribute 'enable_dynamic_creation'}
FUNCTION_BLOCK _ETcVnWorldCoordinateSystem EXTENDS EnumDatatypeBase
VAR
	localData : ETcVnWorldCoordinateSystem;
	activeData : REFERENCE TO ETcVnWorldCoordinateSystem;
	enumBaseDatatype : _DINT(localData);
END_VAR

METHOD PROTECTED SetBaseDatatypeReference
VAR_INPUT
END_VAR
enumBaseDatatype.MakeReferenceTo(activeData);
END_METHOD

PROPERTY PUBLIC Address : PVOID
GET
Address := ADR(activeData);
END_GET
END_PROPERTY

METHOD PUBLIC ClearReference
VAR_INPUT
END_VAR
activeData REF= localData;
SetBaseDatatypeReference();
END_METHOD

PROPERTY PUBLIC Size : UDINT
GET
Size := SIZEOF(activeData);
END_GET
END_PROPERTY

METHOD FB_init : BOOL
VAR_INPUT
	bInitRetains : BOOL; // if TRUE, the retain variables are initialized (warm start / cold start)
	bInCopyCode : BOOL;  // if TRUE, the instance afterwards gets moved into the copy code (online change)
	InitialValue : ETcVnWorldCoordinateSystem;
END_VAR
localData := InitialValue;
AddBaseDatatype(enumBaseDatatype);
ClearReference();

AddLocalEnumeration('TCVN_WCS_X_RIGHT_Y_DOWN' , ETcVnWorldCoordinateSystem.TCVN_WCS_X_RIGHT_Y_DOWN);
AddLocalEnumeration('TCVN_WCS_X_DOWN_Y_RIGHT', ETcVnWorldCoordinateSystem.TCVN_WCS_X_DOWN_Y_RIGHT);
AddLocalEnumeration('TCVN_WCS_X_LEFT_Y_DOWN', ETcVnWorldCoordinateSystem.TCVN_WCS_X_LEFT_Y_DOWN);
AddLocalEnumeration('TCVN_WCS_X_UP_Y_RIGHT', ETcVnWorldCoordinateSystem.TCVN_WCS_X_UP_Y_RIGHT);
AddLocalEnumeration('TCVN_WCS_X_RIGHT_Y_UP', ETcVnWorldCoordinateSystem.TCVN_WCS_X_RIGHT_Y_UP);
AddLocalEnumeration('TCVN_WCS_X_DOWN_Y_LEFT', ETcVnWorldCoordinateSystem.TCVN_WCS_X_DOWN_Y_LEFT);
AddLocalEnumeration('TCVN_WCS_X_LEFT_Y_UP', ETcVnWorldCoordinateSystem.TCVN_WCS_X_LEFT_Y_UP);
AddLocalEnumeration('TCVN_WCS_X_UP_Y_LEFT', ETcVnWorldCoordinateSystem.TCVN_WCS_X_UP_Y_LEFT);
END_METHOD

METHOD PRIVATE AddLocalEnumeration
VAR_INPUT
	Enumeration : T_MAXSTRING;
	Value : ETcVnWorldCoordinateSystem;
END_VAR
AddEnumeration(Enumeration, Value);
END_METHOD

METHOD IsEnumeratorValueEqual : BOOL
VAR_INPUT
	Enumerator : I_KeyValueForwardEnumerator;
END_VAR
VAR
	storedValue : ETcVnWorldCoordinateSystem;
END_VAR
IF NOT Enumerator.TryGet(storedValue) THEN
	RETURN;
END_IF

IsEnumeratorValueEqual := storedValue = activeData;
END_METHOD

METHOD PUBLIC Clone : I_Datatype
VAR
    pClone : POINTER TO _ETcVnWorldCoordinateSystem;
END_VAR
pClone := __NEW(_ETcVnWorldCoordinateSystem(InitialValue := Value));
Clone := pClone^;
END_METHOD

PROPERTY PUBLIC Identifier : T_MAXSTRING
GET
Identifier := 'ETcVnWorldCoordinateSystem';
END_GET
END_PROPERTY

METHOD PUBLIC MakeReferenceTo
VAR_INPUT
	ReferenceTarget : REFERENCE TO ETcVnWorldCoordinateSystem;
END_VAR
activeData REF= ReferenceTarget;
SetBaseDatatypeReference();
END_METHOD

METHOD TryMakeReferenceTo : BOOL
VAR_INPUT
	Target : I_Datatype;
END_VAR
VAR
	pTargetData : POINTER TO ETcVnWorldCoordinateSystem;
END_VAR
IF NOT IsEquivalentTo(Target) THEN
	RETURN;
END_IF

pTargetData := Target.Address;
activeData REF= pTargetData^;
SetBaseDatatypeReference();
TryMakeReferenceTo := TRUE;
END_METHOD

PROPERTY PUBLIC Value : ETcVnWorldCoordinateSystem
GET
Value := activeData;
END_GET
SET
activeData := Value;
END_SET
END_PROPERTY

END_FUNCTION_BLOCK

// Datatypes/Enums/_ETcWatchdogAccumulationType
{attribute 'linkalways'} 
{attribute 'no_explicit_call' := 'This FB is a CLASS and must be accessed using methods or properties'}
{attribute 'enable_dynamic_creation'}
FUNCTION_BLOCK _ETcWatchdogAccumulationType EXTENDS EnumDatatypeBase
VAR
	localData : ETcWatchdogAccumulationType;
	activeData : REFERENCE TO ETcWatchdogAccumulationType;
	enumBaseDatatype : _UINT(localData);
END_VAR

METHOD PROTECTED SetBaseDatatypeReference
VAR_INPUT
END_VAR
enumBaseDatatype.MakeReferenceTo(activeData);
END_METHOD

PROPERTY PUBLIC Address : PVOID
GET
Address := ADR(activeData);
END_GET
END_PROPERTY

METHOD PUBLIC ClearReference
VAR_INPUT
END_VAR
activeData REF= localData;
SetBaseDatatypeReference();
END_METHOD

PROPERTY PUBLIC Size : UDINT
GET
Size := SIZEOF(activeData);
END_GET
END_PROPERTY

METHOD FB_init : BOOL
VAR_INPUT
	bInitRetains : BOOL; // if TRUE, the retain variables are initialized (warm start / cold start)
	bInCopyCode : BOOL;  // if TRUE, the instance afterwards gets moved into the copy code (online change)
	InitialValue : ETcWatchdogAccumulationType;
END_VAR
localData := InitialValue;
AddBaseDatatype(enumBaseDatatype);
ClearReference();

AddLocalEnumeration('WD_ACC_TYPE_MEAN', ETcWatchdogAccumulationType.WD_ACC_TYPE_MEAN);
AddLocalEnumeration('WD_ACC_TYPE_PRODUCT', ETcWatchdogAccumulationType.WD_ACC_TYPE_PRODUCT);
END_METHOD

METHOD PRIVATE AddLocalEnumeration
VAR_INPUT
	Enumeration : T_MAXSTRING;
	Value : ETcWatchdogAccumulationType;
END_VAR
AddEnumeration(Enumeration, Value);
END_METHOD

METHOD IsEnumeratorValueEqual : BOOL
VAR_INPUT
	Enumerator : I_KeyValueForwardEnumerator;
END_VAR
VAR
	storedValue : ETcWatchdogAccumulationType;
END_VAR
IF NOT Enumerator.TryGet(storedValue) THEN
	RETURN;
END_IF

IsEnumeratorValueEqual := storedValue = activeData;
END_METHOD

METHOD PUBLIC Clone : I_Datatype
VAR
    pClone : POINTER TO _ETcWatchdogAccumulationType;
END_VAR
pClone := __NEW(_ETcWatchdogAccumulationType(InitialValue := Value));
Clone := pClone^;
END_METHOD

PROPERTY PUBLIC Identifier : T_MAXSTRING
GET
Identifier := 'ETcWatchdogAccumulationType';
END_GET
END_PROPERTY

METHOD PUBLIC MakeReferenceTo
VAR_INPUT
	ReferenceTarget : REFERENCE TO ETcWatchdogAccumulationType;
END_VAR
activeData REF= ReferenceTarget;
SetBaseDatatypeReference();
END_METHOD

METHOD TryMakeReferenceTo : BOOL
VAR_INPUT
	Target : I_Datatype;
END_VAR
VAR
	pTargetData : POINTER TO ETcWatchdogAccumulationType;
END_VAR
IF NOT IsEquivalentTo(Target) THEN
	RETURN;
END_IF

pTargetData := Target.Address;
activeData REF= pTargetData^;
SetBaseDatatypeReference();
TryMakeReferenceTo := TRUE;
END_METHOD

PROPERTY PUBLIC Value : ETcWatchdogAccumulationType
GET
Value := activeData;
END_GET
SET
activeData := Value;
END_SET
END_PROPERTY

END_FUNCTION_BLOCK

// Datatypes/Enums/_GEV_CAMERA_STATE
{attribute 'linkalways'} 
{attribute 'no_explicit_call' := 'This FB is a CLASS and must be accessed using methods or properties'}
{attribute 'enable_dynamic_creation'}
FUNCTION_BLOCK _GEV_CAMERA_STATE EXTENDS EnumDatatypeBase
VAR
	localData : GEV_CAMERA_STATE;
	activeData : REFERENCE TO GEV_CAMERA_STATE;
	enumBaseDatatype : _BYTE(localData);
END_VAR

METHOD PROTECTED SetBaseDatatypeReference
VAR_INPUT
END_VAR
enumBaseDatatype.MakeReferenceTo(activeData);
END_METHOD

PROPERTY PUBLIC Address : PVOID
GET
Address := ADR(activeData);
END_GET
END_PROPERTY

METHOD PUBLIC ClearReference
VAR_INPUT
END_VAR
activeData REF= localData;
SetBaseDatatypeReference();
END_METHOD

PROPERTY PUBLIC Size : UDINT
GET
Size := SIZEOF(activeData);
END_GET
END_PROPERTY

METHOD FB_init : BOOL
VAR_INPUT
	bInitRetains : BOOL; // if TRUE, the retain variables are initialized (warm start / cold start)
	bInCopyCode : BOOL;  // if TRUE, the instance afterwards gets moved into the copy code (online change)
	InitialValue : GEV_CAMERA_STATE;
END_VAR
localData := InitialValue;
AddBaseDatatype(enumBaseDatatype);
ClearReference();

AddLocalEnumeration('GEV_CAMERA_IDLE', GEV_CAMERA_STATE.GEV_CAMERA_IDLE);
AddLocalEnumeration('GEV_CONTROL_CHANNEL_OPEN_MASK', GEV_CAMERA_STATE.GEV_CONTROL_CHANNEL_OPEN_MASK);
AddLocalEnumeration('GEV_STREAM_CHANNELS_OPEN_MASK', GEV_CAMERA_STATE.GEV_STREAM_CHANNELS_OPEN_MASK);
AddLocalEnumeration('GEV_CONTROL_CHANNEL_OPEN', GEV_CAMERA_STATE.GEV_CONTROL_CHANNEL_OPEN);
AddLocalEnumeration('GEV_STREAM_CHANNELS_OPEN', GEV_CAMERA_STATE.GEV_STREAM_CHANNELS_OPEN);
END_METHOD

METHOD PRIVATE AddLocalEnumeration
VAR_INPUT
	Enumeration : T_MAXSTRING;
	Value : GEV_CAMERA_STATE;
END_VAR
AddEnumeration(Enumeration, Value);
END_METHOD

METHOD IsEnumeratorValueEqual : BOOL
VAR_INPUT
	Enumerator : I_KeyValueForwardEnumerator;
END_VAR
VAR
	storedValue : GEV_CAMERA_STATE;
END_VAR
IF NOT Enumerator.TryGet(storedValue) THEN
	RETURN;
END_IF

IsEnumeratorValueEqual := storedValue = activeData;
END_METHOD

METHOD PUBLIC Clone : I_Datatype
VAR
    pClone : POINTER TO _GEV_CAMERA_STATE;
END_VAR
pClone := __NEW(_GEV_CAMERA_STATE(InitialValue := Value));
Clone := pClone^;
END_METHOD

PROPERTY PUBLIC Identifier : T_MAXSTRING
GET
Identifier := 'GEV_CAMERA_STATE';
END_GET
END_PROPERTY

METHOD PUBLIC MakeReferenceTo
VAR_INPUT
	ReferenceTarget : REFERENCE TO GEV_CAMERA_STATE;
END_VAR
activeData REF= ReferenceTarget;
SetBaseDatatypeReference();
END_METHOD

METHOD TryMakeReferenceTo : BOOL
VAR_INPUT
	Target : I_Datatype;
END_VAR
VAR
	pTargetData : POINTER TO GEV_CAMERA_STATE;
END_VAR
IF NOT IsEquivalentTo(Target) THEN
	RETURN;
END_IF

pTargetData := Target.Address;
activeData REF= pTargetData^;
SetBaseDatatypeReference();
TryMakeReferenceTo := TRUE;
END_METHOD

PROPERTY PUBLIC Value : GEV_CAMERA_STATE
GET
Value := activeData;
END_GET
SET
activeData := Value;
END_SET
END_PROPERTY

END_FUNCTION_BLOCK

// Datatypes/Interfaces/_ITcVnContainer
{attribute 'linkalways'} 
{attribute 'no_explicit_call' := 'This FB is a CLASS and must be accessed using methods or properties'}
{attribute 'enable_dynamic_creation'}
FUNCTION_BLOCK _ITcVnContainer EXTENDS InterfaceDatatypeBase
VAR
	localData : ITcVnContainer;
	activeData : REFERENCE TO ITcVnContainer REF= localData;
END_VAR

PROPERTY PUBLIC Address : PVOID
GET
Address := ADR(activeData);
END_GET
END_PROPERTY

METHOD PUBLIC ClearReference
VAR_INPUT
END_VAR
activeData REF= localData;
END_METHOD

PROPERTY PUBLIC Size : UDINT
GET
Size := SIZEOF(activeData);
END_GET
END_PROPERTY

METHOD FB_exit : BOOL
VAR_INPUT
	bInCopyCode : BOOL; // if TRUE, the exit method is called for exiting an instance that is copied afterwards (online change).
END_VAR
IF bInCopyCode THEN
	RETURN;
END_IF

TryTcReleaseLocal();
END_METHOD

METHOD PRIVATE Serialize_ContainerType_Vector_DINT
VAR_INPUT
	Serializer : I_Serializer;
END_VAR
VAR
	hr : HRESULT;
	_value : _DINT(0);
	elementCount : ULINT;
	i : ULINT;
END_VAR
activeData.GetElementNum(elementCount);

FOR i := 0 TO elementCount - 1 DO 
	
	hr := F_VN_GetAt_DINT(activeData, _value.Value, i, S_OK);
	
	IF SUCCEEDED(hr) THEN
		Serializer.AddObject(_value);
	ELSE
		Serializer.AddNull();
	END_IF
	
END_FOR
END_METHOD

METHOD PRIVATE Serialize_ContainerType_Vector_INT
VAR_INPUT
	Serializer : I_Serializer;
END_VAR
VAR
	hr : HRESULT;
	_value : _INT(0);
	elementCount : ULINT;
	i : ULINT;
END_VAR
activeData.GetElementNum(elementCount);

FOR i := 0 TO elementCount - 1 DO 
	
	hr := F_VN_GetAt_INT(activeData, _value.Value, i, S_OK);
	
	IF SUCCEEDED(hr) THEN
		Serializer.AddObject(_value);
	ELSE
		Serializer.AddNull();
	END_IF
	
END_FOR
END_METHOD

METHOD PRIVATE Serialize_ContainerType_Vector_ITcVnImage
VAR_INPUT
	Serializer : I_Serializer;
END_VAR
VAR
	hr : HRESULT;
	_value : _ITcVnImage;
	elementCount : ULINT;
	i : ULINT;
END_VAR
activeData.GetElementNum(elementCount);

FOR i := 0 TO elementCount - 1 DO 
	
	hr := F_VN_GetAt_ITcVnImage(activeData, _value.Value, i, S_OK);
	
	IF SUCCEEDED(hr) THEN
		Serializer.AddObject(_value);
	ELSE
		Serializer.AddNull();
	END_IF
	
END_FOR
END_METHOD

METHOD PRIVATE Serialize_ContainerType_Vector_LREAL
VAR_INPUT
	Serializer : I_Serializer;
END_VAR
VAR
	hr : HRESULT;
	_value : _LREAL(0);
	elementCount : ULINT;
	i : ULINT;
END_VAR
activeData.GetElementNum(elementCount);

FOR i := 0 TO elementCount - 1 DO 
	
	hr := F_VN_GetAt_LREAL(activeData, _value.Value, i, S_OK);
	
	IF SUCCEEDED(hr) THEN
		Serializer.AddObject(_value);
	ELSE
		Serializer.AddNull();
	END_IF
	
END_FOR
END_METHOD

METHOD PRIVATE Serialize_ContainerType_Vector_REAL
VAR_INPUT
	Serializer : I_Serializer;
END_VAR
VAR
	hr : HRESULT;
	_value : _REAL(0);
	elementCount : ULINT;
	i : ULINT;
END_VAR
activeData.GetElementNum(elementCount);

FOR i := 0 TO elementCount - 1 DO 
	
	hr := F_VN_GetAt_REAL(activeData, _value.Value, i, S_OK);
	
	IF SUCCEEDED(hr) THEN
		Serializer.AddObject(_value);
	ELSE
		Serializer.AddNull();
	END_IF
	
END_FOR
END_METHOD

METHOD PRIVATE Serialize_ContainerType_Vector_SINT
VAR_INPUT
	Serializer : I_Serializer;
END_VAR
VAR
	hr : HRESULT;
	_value : _SINT(0);
	elementCount : ULINT;
	i : ULINT;
END_VAR
activeData.GetElementNum(elementCount);

FOR i := 0 TO elementCount - 1 DO 
	
	hr := F_VN_GetAt_SINT(activeData, _value.Value, i, S_OK);
	
	IF SUCCEEDED(hr) THEN
		Serializer.AddObject(_value);
	ELSE
		Serializer.AddNull();
	END_IF
	
END_FOR
END_METHOD

METHOD PRIVATE Serialize_ContainerType_Vector_UDINT
VAR_INPUT
	Serializer : I_Serializer;
END_VAR
VAR
	hr : HRESULT;
	_value : _ULINT(0);
	elementCount : ULINT;
	i : ULINT;
END_VAR
activeData.GetElementNum(elementCount);

FOR i := 0 TO elementCount - 1 DO 
	
	hr := F_VN_GetAt_ULINT(activeData, _value.Value, i, S_OK);
	
	IF SUCCEEDED(hr) THEN
		Serializer.AddObject(_value);
	ELSE
		Serializer.AddNull();
	END_IF
	
END_FOR
END_METHOD

METHOD PRIVATE Serialize_ContainerType_Vector_UINT
VAR_INPUT
	Serializer : I_Serializer;
END_VAR
VAR
	hr : HRESULT;
	_value : _UINT(0);
	elementCount : ULINT;
	i : ULINT;
END_VAR
activeData.GetElementNum(elementCount);

FOR i := 0 TO elementCount - 1 DO 
	
	hr := F_VN_GetAt_UINT(activeData, _value.Value, i, S_OK);
	
	IF SUCCEEDED(hr) THEN
		Serializer.AddObject(_value);
	ELSE
		Serializer.AddNull();
	END_IF
	
END_FOR
END_METHOD

METHOD PRIVATE Serialize_ContainerType_Vector_ULINT
VAR_INPUT
	Serializer : I_Serializer;
END_VAR
VAR
	hr : HRESULT;
	_value : _ULINT(0);
	elementCount : ULINT;
	i : ULINT;
END_VAR
activeData.GetElementNum(elementCount);

FOR i := 0 TO elementCount - 1 DO 
	
	hr := F_VN_GetAt_ULINT(activeData, _value.Value, i, S_OK);
	
	IF SUCCEEDED(hr) THEN
		Serializer.AddObject(_value);
	ELSE
		Serializer.AddNull();
	END_IF
	
END_FOR
END_METHOD

METHOD PRIVATE Serialize_ContainerType_Vector_USINT
VAR_INPUT
	Serializer : I_Serializer;
END_VAR
VAR
	hr : HRESULT;
	_value : _USINT(0);
	elementCount : ULINT;
	i : ULINT;
END_VAR
activeData.GetElementNum(elementCount);

FOR i := 0 TO elementCount - 1 DO 
	
	hr := F_VN_GetAt_USINT(activeData, _value.Value, i, S_OK);
	
	IF SUCCEEDED(hr) THEN
		Serializer.AddObject(_value);
	ELSE
		Serializer.AddNull();
	END_IF
	
END_FOR
END_METHOD

METHOD PUBLIC TryTcReleaseLocal : BOOL
VAR_INPUT
END_VAR
IF localData = 0 THEN
	RETURN;
END_IF

IF localData.TcRelease() = 0 THEN
	localData := 0;
END_IF

TryTcReleaseLocal := TRUE;
END_METHOD

METHOD PUBLIC Clone : I_Datatype
VAR
    pClone : POINTER TO _ITcVnContainer;
END_VAR
pClone := __NEW(_ITcVnContainer);
Clone := pClone^;
END_METHOD

PROPERTY PUBLIC Identifier : T_MAXSTRING
GET
Identifier := 'ITcVnContainer';
END_GET
END_PROPERTY

METHOD PUBLIC MakeReferenceTo
VAR_INPUT
	ReferenceTarget : REFERENCE TO ITcVnContainer;
END_VAR
activeData REF= ReferenceTarget;
END_METHOD

METHOD PUBLIC SerializeWith
VAR_INPUT
	Serializer : I_Serializer;
END_VAR
VAR
	containerTypeName : _STRING('');
	containerTypeGuid : _GUID;
	elementTypeGuid : _GUID;
    elementNum : _ULINT(0);
    elementSize : _ULINT(0);
END_VAR
IF NOT (activeData <> 0) THEN
	Serializer.AddNull();
	RETURN;
END_IF

activeData.GetTypeName(containerTypeName.Value,UDINT_TO_UINT(containerTypeName.Size));
activeData.GetTypeGuid(containerTypeGuid.Value);
activeData.GetElementTypeGuid(elementTypeGuid.Value);
activeData.GetElementNum(elementNum.Value);
activeData.GetElementSize(elementSize.Value);

Serializer.StartObject();
Serializer.AddKeyObject('containerTypeName', containerTypeName);
Serializer.AddKeyString('containerTypeGuid', containerTypeGuid.ToString());
Serializer.AddKeyString('elementTypeGuid', elementTypeGuid.ToString());
Serializer.AddKeyObject('elementNum', elementNum);
Serializer.AddKeyObject('elementSize', elementSize);
Serializer.AddKey('elements');
Serializer.StartArray();

IF containerTypeName.Value = 'CTcVnContainer_Vector_SINT' THEN
	Serialize_ContainerType_Vector_SINT(Serializer);		
ELSIF containerTypeName.Value = 'CTcVnContainer_Vector_USINT' THEN
	Serialize_ContainerType_Vector_USINT(Serializer);
ELSIF containerTypeName.Value = 'CTcVnContainer_Vector_INT' THEN
	Serialize_ContainerType_Vector_INT(Serializer);
ELSIF containerTypeName.Value = 'CTcVnContainer_Vector_UINT' THEN
	Serialize_ContainerType_Vector_UINT(Serializer);
ELSIF containerTypeName.Value = 'CTcVnContainer_Vector_DINT' THEN
	Serialize_ContainerType_Vector_DINT(Serializer);
ELSIF containerTypeName.Value = 'CTcVnContainer_Vector_UDINT' THEN
	Serialize_ContainerType_Vector_UDINT(Serializer);
ELSIF containerTypeName.Value = 'CTcVnContainer_Vector_ULINT' THEN
	Serialize_ContainerType_Vector_ULINT(Serializer);
ELSIF containerTypeName.Value = 'CTcVnContainer_Vector_REAL' THEN
	Serialize_ContainerType_Vector_REAL(Serializer);
ELSIF containerTypeName.Value = 'CTcVnContainer_Vector_LREAL' THEN
	Serialize_ContainerType_Vector_LREAL(Serializer);
ELSIF containerTypeName.Value = 'CTcVnContainer_Vector_ITcVnImage' THEN
	Serialize_ContainerType_Vector_ITcVnImage(Serializer);
//ELSIF containerTypeName.Value = 'CTcVnContainer_Vector_' THEN
//	Serialize_ContainerType_Vector_(Serializer);
//ELSIF containerTypeName.Value = 'CTcVnContainer_Vector_' THEN
//	Serialize_ContainerType_Vector_(Serializer);
//ELSIF containerTypeName.Value = 'CTcVnContainer_Vector_' THEN
//	Serialize_ContainerType_Vector_(Serializer);
//ELSIF containerTypeName.Value = 'CTcVnContainer_Vector_' THEN
//	Serialize_ContainerType_Vector_(Serializer);
//ELSIF containerTypeName.Value = 'CTcVnContainer_Vector_' THEN
//	Serialize_ContainerType_Vector_(Serializer);
//ELSIF containerTypeName.Value = 'CTcVnContainer_Vector_' THEN
//	Serialize_ContainerType_Vector_(Serializer);	
		
END_IF
Serializer.EndArray();
Serializer.EndObject();
END_METHOD

METHOD TryDeserializeFrom : BOOL
VAR_INPUT
	Deserializer : I_Deserializer;
	Feedback : I_DeserializerFeedback;
END_VAR
VAR
END_VAR
// not yet implemented.  This will just be a reverse of the serialization code.
END_METHOD

METHOD TryMakeReferenceTo : BOOL
VAR_INPUT
	Target : I_Datatype;
END_VAR
VAR
	pTargetData : POINTER TO ITcVnContainer;
END_VAR
IF NOT IsEquivalentTo(Target) THEN
	RETURN;
END_IF

pTargetData := Target.Address;
activeData REF= pTargetData^;
TryMakeReferenceTo := TRUE;
END_METHOD

PROPERTY PUBLIC Value : REFERENCE TO ITcVnContainer
GET
Value REF= activeData;
END_GET
END_PROPERTY

METHOD PUBLIC HasType : BOOL
VAR_INPUT
	Expected : STRING;
END_VAR
VAR
    name : STRING;
END_VAR
IF NOT TryGetTypeName(name) THEN
    RETURN;
END_IF

IF NOT (Expected = name) THEN
    RETURN;
END_IF

HasType := TRUE;
END_METHOD

PROPERTY PUBLIC IsValid : BOOL
GET
IsValid := activeData <> 0;
END_GET
END_PROPERTY

METHOD PUBLIC TryGetTypeName : BOOL
VAR_INPUT
	Destination : REFERENCE TO STRING;
END_VAR
IF NOT IsValid THEN
	RETURN;
END_IF

TryGetTypeName := SUCCEEDED(activeData.GetTypeName(Destination, 255));
END_METHOD

METHOD PUBLIC TryTcAddRef : BOOL
VAR_INPUT
END_VAR
IF activeData = 0 THEN
	RETURN;
END_IF

IF activeData.TcAddRef() = 0 THEN
	activeData := 0;
END_IF

TryTcAddRef := TRUE;
END_METHOD

METHOD PUBLIC TryTcRelease : BOOL
VAR_INPUT
END_VAR
IF activeData = 0 THEN
	RETURN;
END_IF

IF activeData.TcRelease() = 0 THEN
	activeData := 0;
END_IF

TryTcRelease := TRUE;
END_METHOD

END_FUNCTION_BLOCK

// Datatypes/Structs/_TcVnCircularArc
{attribute 'linkalways'} 
{attribute 'no_explicit_call' := 'This FB is a CLASS and must be accessed using methods or properties'}
{attribute 'enable_dynamic_creation'}
FUNCTION_BLOCK _TcVnCircularArc EXTENDS StructuredDatatypeBase
VAR
	localData : TcVnCircularArc;
	activeData : REFERENCE TO TcVnCircularArc REF= localData;
    _aCenter : _TcVnPoint2_REAL();
    _fRadius : _REAL(localdata.fRadius);
    _fStartAngle : _REAL(localdata.fStartAngle);
    _fEndAngle : _REAL(localdata.fEndAngle);
END_VAR

PROPERTY PUBLIC Address : PVOID
GET
Address := ADR(activeData);
END_GET
END_PROPERTY

METHOD PUBLIC ClearReference
VAR_INPUT
END_VAR
activeData REF= localData;
SetMemberReference();
END_METHOD

PROPERTY PUBLIC Size : UDINT
GET
Size := SIZEOF(activeData);
END_GET
END_PROPERTY

METHOD FB_init : BOOL
VAR_INPUT
	bInitRetains : BOOL; // if TRUE, the retain variables are initialized (warm start / cold start)
	bInCopyCode : BOOL;  // if TRUE, the instance afterwards gets moved into the copy code (online change)
END_VAR
SetMemberReference();
AddMember('aCenter', _aCenter);
AddMember('fRadius', _fRadius);
AddMember('fStartAngle', _fStartAngle);
AddMember('fEndAngle', _fEndAngle);
END_METHOD

METHOD PROTECTED SetMemberReference
VAR_INPUT
END_VAR
_aCenter.MakeReferenceTo(activeData.aCenter);
_fRadius.MakeReferenceTo(activeData.fRadius);
_fStartAngle.MakeReferenceTo(activeData.fStartAngle);
_fEndAngle.MakeReferenceTo(activeData.fEndAngle);
END_METHOD

METHOD PUBLIC Clone : I_Datatype
VAR
    pClone : POINTER TO _TcVnCircularArc;
END_VAR
pClone := __NEW(_TcVnCircularArc());
pClone^.Value := Value;
Clone := pClone^;
END_METHOD

PROPERTY PUBLIC Identifier : T_MAXSTRING
GET
Identifier := 'TcVnCircularArc';
END_GET
END_PROPERTY

METHOD PUBLIC MakeReferenceTo
VAR_INPUT
	ReferenceTarget : REFERENCE TO TcVnCircularArc;
END_VAR
activeData REF= ReferenceTarget;
SetMemberReference();
END_METHOD

METHOD TryMakeReferenceTo : BOOL
VAR_INPUT
	Target : I_Datatype;
END_VAR
VAR
	pTargetData : POINTER TO TcVnCircularArc;
END_VAR
IF NOT IsEquivalentTo(Target) THEN
	RETURN;
END_IF

pTargetData := Target.Address;
activeData REF= pTargetData^;
SetMemberReference();
TryMakeReferenceTo := TRUE;
END_METHOD

PROPERTY PUBLIC Value : REFERENCE TO TcVnCircularArc
GET
Value REF= activeData;
END_GET
END_PROPERTY

PROPERTY PUBLIC aCenter : REFERENCE TO _TcVnPoint2_REAL
GET
aCenter REF= _aCenter;
END_GET
END_PROPERTY

PROPERTY PUBLIC fEndAngle : REFERENCE TO _REAL
GET
fEndAngle REF= _fEndAngle;
END_GET
END_PROPERTY

PROPERTY PUBLIC fRadius : REFERENCE TO _REAL
GET
fRadius REF= _fRadius;
END_GET
END_PROPERTY

PROPERTY PUBLIC fStartAngle : REFERENCE TO _REAL
GET
fStartAngle REF= _fStartAngle;
END_GET
END_PROPERTY

END_FUNCTION_BLOCK

// Datatypes/Structs/_TcVnDMatch
{attribute 'linkalways'} 
{attribute 'no_explicit_call' := 'This FB is a CLASS and must be accessed using methods or properties'}
{attribute 'enable_dynamic_creation'}
FUNCTION_BLOCK _TcVnDMatch EXTENDS StructuredDatatypeBase
VAR
	localData : TcVnDMatch;
	activeData : REFERENCE TO TcVnDMatch REF= localData;
    _nQueryIdx : _DINT(localdata.nQueryIdx);
    _nTrainIdx : _DINT(localdata.nTrainIdx);
    _nImageIdx : _DINT(localdata.nImageIdx);
    _fDistance : _REAL(localdata.fDistance);
END_VAR

PROPERTY PUBLIC Address : PVOID
GET
Address := ADR(activeData);
END_GET
END_PROPERTY

METHOD PUBLIC ClearReference
VAR_INPUT
END_VAR
activeData REF= localData;
SetMemberReference();
END_METHOD

PROPERTY PUBLIC Size : UDINT
GET
Size := SIZEOF(activeData);
END_GET
END_PROPERTY

METHOD FB_init : BOOL
VAR_INPUT
	bInitRetains : BOOL; // if TRUE, the retain variables are initialized (warm start / cold start)
	bInCopyCode : BOOL;  // if TRUE, the instance afterwards gets moved into the copy code (online change)
END_VAR
SetMemberReference();
AddMember('nQueryIdx', _nQueryIdx);
AddMember('nTrainIdx', _nTrainIdx);
AddMember('nImageIdx', _nImageIdx);
AddMember('fDistance', _fDistance);
END_METHOD

METHOD PROTECTED SetMemberReference
VAR_INPUT
END_VAR
_nQueryIdx.MakeReferenceTo(activeData.nQueryIdx);
_nTrainIdx.MakeReferenceTo(activeData.nTrainIdx);
_nImageIdx.MakeReferenceTo(activeData.nImageIdx);
_fDistance.MakeReferenceTo(activeData.fDistance);
END_METHOD

METHOD PUBLIC Clone : I_Datatype
VAR
    pClone : POINTER TO _TcVnDMatch;
END_VAR
pClone := __NEW(_TcVnDMatch());
pClone^.Value := Value;
Clone := pClone^;
END_METHOD

PROPERTY PUBLIC Identifier : T_MAXSTRING
GET
Identifier := 'TcVnDMatch';
END_GET
END_PROPERTY

METHOD PUBLIC MakeReferenceTo
VAR_INPUT
	ReferenceTarget : REFERENCE TO TcVnDMatch;
END_VAR
activeData REF= ReferenceTarget;
SetMemberReference();
END_METHOD

METHOD TryMakeReferenceTo : BOOL
VAR_INPUT
	Target : I_Datatype;
END_VAR
VAR
	targetAsStruct : I_StructuredDatatype;
	pTargetData : POINTER TO TcVnDMatch;
END_VAR
IF NOT Target.TryResolveAsStructuredDatatype(targetAsStruct) THEN
	RETURN;
END_IF

IF NOT (targetAsStruct.Identifier = Identifier) THEN
	RETURN;
END_IF

pTargetData := Target.Address;
activeData REF= pTargetData^;
SetMemberReference();
TryMakeReferenceTo := TRUE;
END_METHOD

PROPERTY PUBLIC Value : REFERENCE TO TcVnDMatch
GET
Value REF= activeData;
END_GET
END_PROPERTY

PROPERTY PUBLIC fDistance : REFERENCE TO _REAL
GET
fDistance REF= _fDistance;
END_GET
END_PROPERTY

PROPERTY PUBLIC nImageIdx : REFERENCE TO _DINT
GET
nImageIdx REF= _nImageIdx;
END_GET
END_PROPERTY

PROPERTY PUBLIC nQueryIdx : REFERENCE TO _DINT
GET
nQueryIdx REF= _nQueryIdx;
END_GET
END_PROPERTY

PROPERTY PUBLIC nTrainIdx : REFERENCE TO _DINT
GET
nTrainIdx REF= _nTrainIdx;
END_GET
END_PROPERTY

END_FUNCTION_BLOCK

// Datatypes/Structs/_TcVnKeyPoint
{attribute 'linkalways'} 
{attribute 'no_explicit_call' := 'This FB is a CLASS and must be accessed using methods or properties'}
{attribute 'enable_dynamic_creation'}
FUNCTION_BLOCK _TcVnKeyPoint EXTENDS StructuredDatatypeBase
VAR
	localData : TcVnKeyPoint;
	activeData : REFERENCE TO TcVnKeyPoint REF= localData;
    _aPoint : _TcVnPoint2_REAL();
    _fDiameter : _REAL(localdata.fDiameter);
    _fAngle : _REAL(localdata.fAngle);
    _fResponse : _REAL(localdata.fResponse);
    _nOctave : _DINT(localdata.nOctave);
    _nClassId : _DINT(localdata.nClassId);
END_VAR

PROPERTY PUBLIC Address : PVOID
GET
Address := ADR(activeData);
END_GET
END_PROPERTY

METHOD PUBLIC ClearReference
VAR_INPUT
END_VAR
activeData REF= localData;
SetMemberReference();
END_METHOD

PROPERTY PUBLIC Size : UDINT
GET
Size := SIZEOF(activeData);
END_GET
END_PROPERTY

METHOD FB_init : BOOL
VAR_INPUT
	bInitRetains : BOOL; // if TRUE, the retain variables are initialized (warm start / cold start)
	bInCopyCode : BOOL;  // if TRUE, the instance afterwards gets moved into the copy code (online change)
END_VAR
SetMemberReference();
AddMember('aPoint', _aPoint);
AddMember('fDiameter', _fDiameter);
AddMember('fAngle', _fAngle);
AddMember('fResponse', _fResponse);
AddMember('nOctave', _nOctave);
AddMember('nClassId', _nClassId);
END_METHOD

METHOD PROTECTED SetMemberReference
VAR_INPUT
END_VAR
_aPoint.MakeReferenceTo(activeData.aPoint);
_fDiameter.MakeReferenceTo(activeData.fDiameter);
_fAngle.MakeReferenceTo(activeData.fAngle);
_fResponse.MakeReferenceTo(activeData.fResponse);
_nOctave.MakeReferenceTo(activeData.nOctave);
_nClassId.MakeReferenceTo(activeData.nClassId);
END_METHOD

METHOD PUBLIC Clone : I_Datatype
VAR
    pClone : POINTER TO _TcVnKeyPoint;
END_VAR
pClone := __NEW(_TcVnKeyPoint());
pClone^.Value := Value;
Clone := pClone^;
END_METHOD

PROPERTY PUBLIC Identifier : T_MAXSTRING
GET
Identifier := 'TcVnKeyPoint';
END_GET
END_PROPERTY

METHOD PUBLIC MakeReferenceTo
VAR_INPUT
	ReferenceTarget : REFERENCE TO TcVnKeyPoint;
END_VAR
activeData REF= ReferenceTarget;
SetMemberReference();
END_METHOD

METHOD TryMakeReferenceTo : BOOL
VAR_INPUT
	Target : I_Datatype;
END_VAR
VAR
	pTargetData : POINTER TO TcVnKeyPoint;
END_VAR
IF NOT IsEquivalentTo(Target) THEN
	RETURN;
END_IF

pTargetData := Target.Address;
activeData REF= pTargetData^;
SetMemberReference();
TryMakeReferenceTo := TRUE;
END_METHOD

PROPERTY PUBLIC Value : REFERENCE TO TcVnKeyPoint
GET
Value REF= activeData;
END_GET
END_PROPERTY

PROPERTY PUBLIC aPoint : REFERENCE TO _TcVnPoint2_REAL
GET
aPoint REF= _aPoint;
END_GET
END_PROPERTY

PROPERTY PUBLIC fAngle : REFERENCE TO _REAL
GET
fAngle REF= _fAngle;
END_GET
END_PROPERTY

PROPERTY PUBLIC fDiameter : REFERENCE TO _REAL
GET
fDiameter REF= _fDiameter;
END_GET
END_PROPERTY

PROPERTY PUBLIC fResponse : REFERENCE TO _REAL
GET
fResponse REF= _fResponse;
END_GET
END_PROPERTY

PROPERTY PUBLIC nClassId : REFERENCE TO _DINT
GET
nClassId REF= _nClassId;
END_GET
END_PROPERTY

PROPERTY PUBLIC nOctave : REFERENCE TO _DINT
GET
nOctave REF= _nOctave;
END_GET
END_PROPERTY

END_FUNCTION_BLOCK

// Datatypes/Structs/_TcVnParamsBlobDetection
{attribute 'linkalways'} 
{attribute 'no_explicit_call' := 'This FB is a CLASS and must be accessed using methods or properties'}
{attribute 'enable_dynamic_creation'}
FUNCTION_BLOCK _TcVnParamsBlobDetection EXTENDS StructuredDatatypeBase
VAR
	localData : TcVnParamsBlobDetection;
	activeData : REFERENCE TO TcVnParamsBlobDetection REF= localData;
    _bFilterByArea         : _BOOL(localdata.bFilterByArea);
    _bFilterByCircularity  : _BOOL(localdata.bFilterByCircularity);
    _bFilterByConvexity    : _BOOL(localdata.bFilterByConvexity);
    _bFilterByEccentricity : _BOOL(localdata.bFilterByEccentricity);
    _bFilterByInertiaRatio : _BOOL(localdata.bFilterByInertiaRatio);
    _fMinArea              : _REAL(localdata.fMinArea);
    _fMaxArea              : _REAL(localdata.fMaxArea);
    _fMinCircularity       : _REAL(localdata.fMinCircularity);
    _fMaxCircularity       : _REAL(localdata.fMaxCircularity);
    _fMinConvexity         : _REAL(localdata.fMinConvexity);
    _fMaxConvexity         : _REAL(localdata.fMaxConvexity);
    _fMinEccentricity      : _REAL(localdata.fMinEccentricity);
    _fMaxEccentricity      : _REAL(localdata.fMaxEccentricity);
    _fMinInertiaRatio      : _REAL(localdata.fMinInertiaRatio);
    _fMaxInertiaRatio      : _REAL(localdata.fMaxInertiaRatio);
    _eThresholdType        : _ETcVnThresholdType(localdata.eThresholdType);
    _fMinThreshold         : _REAL(localdata.fMinThreshold);
    _fMaxThreshold         : _REAL(localdata.fMaxThreshold);
    _fThresholdStep        : _REAL(localdata.fThresholdStep);
    _fMinBlobDistance      : _REAL(localdata.fMinBlobDistance);
    _nMinRepeatability     : _UDINT(localdata.nMinRepeatability);
    _eBlobCombination      : _ETcVnBlobCombination(localdata.eBlobCombination);
END_VAR

PROPERTY PUBLIC Address : PVOID
GET
Address := ADR(activeData);
END_GET
END_PROPERTY

METHOD PUBLIC ClearReference
VAR_INPUT
END_VAR
activeData REF= localData;
SetMemberReference();
END_METHOD

PROPERTY PUBLIC Size : UDINT
GET
Size := SIZEOF(activeData);
END_GET
END_PROPERTY

METHOD FB_init : BOOL
VAR_INPUT
	bInitRetains : BOOL; // if TRUE, the retain variables are initialized (warm start / cold start)
	bInCopyCode : BOOL;  // if TRUE, the instance afterwards gets moved into the copy code (online change)
END_VAR
SetMemberReference();
AddMember('bFilterByArea', _bFilterByArea);
AddMember('bFilterByCircularity', _bFilterByCircularity);
AddMember('bFilterByConvexity', _bFilterByConvexity);
AddMember('bFilterByEccentricity', _bFilterByEccentricity);
AddMember('bFilterByInertiaRatio', _bFilterByInertiaRatio);
AddMember('fMinArea', _fMinArea);
AddMember('fMaxArea', _fMaxArea);
AddMember('fMinCircularity', _fMinCircularity);
AddMember('fMaxCircularity', _fMaxCircularity);
AddMember('fMinConvexity', _fMinConvexity);
AddMember('fMaxConvexity', _fMaxConvexity);
AddMember('fMinEccentricity', _fMinEccentricity);
AddMember('fMaxEccentricity', _fMaxEccentricity);
AddMember('fMinInertiaRatio', _fMinInertiaRatio);
AddMember('fMaxInertiaRatio', _fMaxInertiaRatio);
AddMember('eThresholdType', _eThresholdType);
AddMember('fMinThreshold', _fMinThreshold);
AddMember('fMaxThreshold', _fMaxThreshold);
AddMember('fThresholdStep',  _fThresholdStep);
AddMember('fMinBlobDistance', _fMinBlobDistance);
AddMember('nMinRepeatability', _nMinRepeatability);
AddMember('eBlobCombination', _eBlobCombination);
END_METHOD

METHOD PROTECTED SetMemberReference
VAR_INPUT
END_VAR
_bFilterByArea.MakeReferenceTo(activeData.bFilterByArea);
_bFilterByCircularity.MakeReferenceTo(activeData.bFilterByCircularity);
_bFilterByConvexity.MakeReferenceTo(activeData.bFilterByConvexity);
_bFilterByEccentricity.MakeReferenceTo(activeData.bFilterByEccentricity);
_bFilterByInertiaRatio.MakeReferenceTo(activeData.bFilterByInertiaRatio);
_fMinArea.MakeReferenceTo(activeData.fMinArea);
_fMaxArea.MakeReferenceTo(activeData.fMaxArea);
_fMinCircularity.MakeReferenceTo(activeData.fMinCircularity);
_fMaxCircularity.MakeReferenceTo(activeData.fMaxCircularity);
_fMinConvexity.MakeReferenceTo(activeData.fMinConvexity);
_fMaxConvexity.MakeReferenceTo(activeData.fMaxConvexity);
_fMinEccentricity.MakeReferenceTo(activeData.fMinEccentricity);
_fMaxEccentricity.MakeReferenceTo(activeData.fMaxEccentricity);
_fMinInertiaRatio.MakeReferenceTo(activeData.fMinInertiaRatio);
_fMaxInertiaRatio.MakeReferenceTo(activeData.fMaxInertiaRatio);
_eThresholdType.MakeReferenceTo(activeData.eThresholdType);
_fMinThreshold.MakeReferenceTo(activeData.fMinThreshold);
_fMaxThreshold.MakeReferenceTo(activeData.fMaxThreshold);
_fThresholdStep.MakeReferenceTo(activeData.fThresholdStep);
_fMinBlobDistance.MakeReferenceTo(activeData.fMinBlobDistance);
_nMinRepeatability.MakeReferenceTo(activeData.nMinRepeatability);
_eBlobCombination.MakeReferenceTo(activeData.eBlobCombination);
END_METHOD

METHOD PUBLIC Clone : I_Datatype
VAR
    pClone : POINTER TO _TcVnParamsBlobDetection;
END_VAR
pClone := __NEW(_TcVnParamsBlobDetection());
pClone^.Value := Value;
Clone := pClone^;
END_METHOD

PROPERTY PUBLIC Identifier : T_MAXSTRING
GET
Identifier := 'TcVnParamsBlobDetection';
END_GET
END_PROPERTY

METHOD PUBLIC MakeReferenceTo
VAR_INPUT
	ReferenceTarget : REFERENCE TO TcVnParamsBlobDetection;
END_VAR
activeData REF= ReferenceTarget;
SetMemberReference();
END_METHOD

METHOD TryMakeReferenceTo : BOOL
VAR_INPUT
	Target : I_Datatype;
END_VAR
VAR
	pTargetData : POINTER TO TcVnParamsBlobDetection;
END_VAR
IF NOT IsEquivalentTo(Target) THEN
	RETURN;
END_IF

pTargetData := Target.Address;
activeData REF= pTargetData^;
SetMemberReference();
TryMakeReferenceTo := TRUE;
END_METHOD

PROPERTY PUBLIC Value : REFERENCE TO TcVnParamsBlobDetection
GET
Value REF= activeData;
END_GET
END_PROPERTY

PROPERTY PUBLIC bFilterByArea : REFERENCE TO _BOOL
GET
bFilterByArea REF= _bFilterByArea;
END_GET
END_PROPERTY

PROPERTY PUBLIC bFilterByCircularity : REFERENCE TO _BOOL
GET
bFilterByCircularity REF= _bFilterByCircularity;
END_GET
END_PROPERTY

PROPERTY PUBLIC bFilterByConvexity : REFERENCE TO _BOOL
GET
bFilterByConvexity REF= _bFilterByConvexity;
END_GET
END_PROPERTY

PROPERTY PUBLIC bFilterByEccentricity : REFERENCE TO _BOOL
GET
bFilterByEccentricity REF= _bFilterByEccentricity;
END_GET
END_PROPERTY

PROPERTY PUBLIC bFilterByInertiaRatio : REFERENCE TO _BOOL
GET
bFilterByInertiaRatio REF= _bFilterByInertiaRatio;
END_GET
END_PROPERTY

PROPERTY PUBLIC eBlobCombination : REFERENCE TO _ETcVnBlobCombination
GET
eBlobCombination REF= _eBlobCombination;
END_GET
END_PROPERTY

PROPERTY PUBLIC eThresholdType : REFERENCE TO _ETcVnThresholdType
GET
eThresholdType REF= _eThresholdType;
END_GET
END_PROPERTY

PROPERTY PUBLIC fMaxArea : REFERENCE TO _REAL
GET
fMaxArea REF= _fMaxArea;
END_GET
END_PROPERTY

PROPERTY PUBLIC fMaxCircularity : REFERENCE TO _REAL
GET
fMaxCircularity REF= _fMaxCircularity;
END_GET
END_PROPERTY

PROPERTY PUBLIC fMaxConvexity : REFERENCE TO _REAL
GET
fMaxConvexity REF= _fMaxConvexity;
END_GET
END_PROPERTY

PROPERTY PUBLIC fMaxEccentricity : REFERENCE TO _REAL
GET
fMaxEccentricity REF= _fMaxEccentricity;
END_GET
END_PROPERTY

PROPERTY PUBLIC fMaxInertiaRatio : REFERENCE TO _REAL
GET
fMaxInertiaRatio REF= _fMaxInertiaRatio;
END_GET
END_PROPERTY

PROPERTY PUBLIC fMaxThreshold : REFERENCE TO _REAL
GET
fMaxThreshold REF= _fMaxThreshold;
END_GET
END_PROPERTY

PROPERTY PUBLIC fMinArea : REFERENCE TO _REAL
GET
fMinArea REF= _fMinArea;
END_GET
END_PROPERTY

PROPERTY PUBLIC fMinBlobDistance : REFERENCE TO _REAL
GET
fMinBlobDistance REF= _fMinBlobDistance;
END_GET
END_PROPERTY

PROPERTY PUBLIC fMinCircularity : REFERENCE TO _REAL
GET
fMinCircularity REF= _fMinCircularity;
END_GET
END_PROPERTY

PROPERTY PUBLIC fMinConvexity : REFERENCE TO _REAL
GET
fMinConvexity REF= _fMinConvexity;
END_GET
END_PROPERTY

PROPERTY PUBLIC fMinEccentricity : REFERENCE TO _REAL
GET
fMinEccentricity REF= _fMinEccentricity;
END_GET
END_PROPERTY

PROPERTY PUBLIC fMinInertiaRatio : REFERENCE TO _REAL
GET
fMinInertiaRatio REF= _fMinInertiaRatio;
END_GET
END_PROPERTY

PROPERTY PUBLIC fMinThreshold : REFERENCE TO _REAL
GET
fMinThreshold REF= _fMinThreshold;
END_GET
END_PROPERTY

PROPERTY PUBLIC fThresholdStep : REFERENCE TO _REAL
GET
fThresholdStep REF= _fThresholdStep;
END_GET
END_PROPERTY

PROPERTY PUBLIC nMinRepeatability : REFERENCE TO _UDINT
GET
nMinRepeatability REF= _nMinRepeatability;
END_GET
END_PROPERTY

END_FUNCTION_BLOCK

// Datatypes/Structs/_TcVnRectangle_UDINT
{attribute 'linkalways'} 
{attribute 'no_explicit_call' := 'This FB is a CLASS and must be accessed using methods or properties'}
{attribute 'enable_dynamic_creation'}
FUNCTION_BLOCK _TcVnRectangle_UDINT EXTENDS StructuredDatatypeBase
VAR
	localData : TcVnRectangle_UDINT;
	activeData : REFERENCE TO TcVnRectangle_UDINT REF= localData;
	_nX : _UDINT(localData.nX);
	_nY : _UDINT(localData.nY);
    _nWidth : _UDINT(localData.nWidth);
	_nHeight : _UDINT(localData.nHeight);
END_VAR

PROPERTY PUBLIC Address : PVOID
GET
Address := ADR(activeData);
END_GET
END_PROPERTY

METHOD PUBLIC ClearReference
VAR_INPUT
END_VAR
activeData REF= localData;
SetMemberReference();
END_METHOD

PROPERTY PUBLIC Size : UDINT
GET
Size := SIZEOF(activeData);
END_GET
END_PROPERTY

METHOD FB_init : BOOL
VAR_INPUT
	bInitRetains : BOOL; // if TRUE, the retain variables are initialized (warm start / cold start)
	bInCopyCode : BOOL;  // if TRUE, the instance afterwards gets moved into the copy code (online change)
END_VAR
SetMemberReference();
AddMember('nX',_nX);
AddMember('nY',_nY);
AddMember('nWidth',_nWidth);
AddMember('nHeight',_nHeight);
END_METHOD

METHOD PROTECTED SetMemberReference
VAR_INPUT
END_VAR
_nX.MakeReferenceTo(activeData.nX);
_nY.MakeReferenceTo(activeData.nY);
_nWidth.MakeReferenceTo(activeData.nWidth);
_nHeight.MakeReferenceTo(activeData.nHeight);
END_METHOD

METHOD PUBLIC Clone : I_Datatype
VAR
    pClone : POINTER TO _TcVnRectangle_UDINT;
END_VAR
pClone := __NEW(_TcVnRectangle_UDINT());
pClone^.Value := Value;
Clone := pClone^;
END_METHOD

PROPERTY PUBLIC Identifier : T_MAXSTRING
GET
Identifier := 'TcVnRectangle_UDINT';
END_GET
END_PROPERTY

METHOD PUBLIC MakeReferenceTo
VAR_INPUT
	ReferenceTarget : REFERENCE TO TcVnRectangle_UDINT;
END_VAR
activeData REF= ReferenceTarget;
SetMemberReference();
END_METHOD

METHOD TryMakeReferenceTo : BOOL
VAR_INPUT
	Target : I_Datatype;
END_VAR
VAR
	pTargetData : POINTER TO TcVnRectangle_UDINT;
END_VAR
IF NOT IsEquivalentTo(Target) THEN
	RETURN;
END_IF

pTargetData := Target.Address;
activeData REF= pTargetData^;
SetMemberReference();
TryMakeReferenceTo := TRUE;
END_METHOD

PROPERTY PUBLIC Value : REFERENCE TO TcVnRectangle_UDINT
GET
Value REF= activeData;
END_GET
END_PROPERTY

PROPERTY PUBLIC nHeight : REFERENCE TO _UDINT
GET
nHeight REF= _nHeight;
END_GET
END_PROPERTY

PROPERTY PUBLIC nWidth : REFERENCE TO _UDINT
GET
nWidth REF= _nWidth;
END_GET
END_PROPERTY

PROPERTY PUBLIC nX : REFERENCE TO _UDINT
GET
nX REF= _nX;
END_GET
END_PROPERTY

PROPERTY PUBLIC nY : REFERENCE TO _UDINT
GET
nY REF= _nY;
END_GET
END_PROPERTY

END_FUNCTION_BLOCK

// Datatypes/Structs/_TcVnRotatedRectangle
{attribute 'linkalways'} 
{attribute 'no_explicit_call' := 'This FB is a CLASS and must be accessed using methods or properties'}
{attribute 'enable_dynamic_creation'}
FUNCTION_BLOCK _TcVnRotatedRectangle EXTENDS StructuredDatatypeBase
VAR
	localData : TcVnRotatedRectangle;
	activeData : REFERENCE TO TcVnRotatedRectangle REF= localData;
    _aCenter : _TcVnPoint2_REAL();
    _stSize : _TcVnSize2_REAL();
    _fAngle : _REAL(localdata.fAngle);
END_VAR

PROPERTY PUBLIC Address : PVOID
GET
Address := ADR(activeData);
END_GET
END_PROPERTY

METHOD PUBLIC ClearReference
VAR_INPUT
END_VAR
activeData REF= localData;
SetMemberReference();
END_METHOD

PROPERTY PUBLIC Size : UDINT
GET
Size := SIZEOF(activeData);
END_GET
END_PROPERTY

METHOD FB_init : BOOL
VAR_INPUT
	bInitRetains : BOOL; // if TRUE, the retain variables are initialized (warm start / cold start)
	bInCopyCode : BOOL;  // if TRUE, the instance afterwards gets moved into the copy code (online change)
END_VAR
SetMemberReference();
AddMember('aCenter', _aCenter);
AddMember('stSize', _stSize);
AddMember('fAngle', _fAngle);
END_METHOD

METHOD PROTECTED SetMemberReference
VAR_INPUT
END_VAR
_aCenter.MakeReferenceTo(activeData.aCenter);
_stsize.MakeReferenceTo(activeData.stSize);
_fAngle.MakeReferenceTo(activeData.fAngle);
END_METHOD

METHOD PUBLIC Clone : I_Datatype
VAR
    pClone : POINTER TO _TcVnRotatedRectangle;
END_VAR
pClone := __NEW(_TcVnRotatedRectangle());
pClone^.Value := Value;
Clone := pClone^;
END_METHOD

PROPERTY PUBLIC Identifier : T_MAXSTRING
GET
Identifier := 'TcVnRotatedRectangle';
END_GET
END_PROPERTY

METHOD PUBLIC MakeReferenceTo
VAR_INPUT
	ReferenceTarget : REFERENCE TO TcVnRotatedRectangle;
END_VAR
activeData REF= ReferenceTarget;
SetMemberReference();
END_METHOD

METHOD TryMakeReferenceTo : BOOL
VAR_INPUT
	Target : I_Datatype;
END_VAR
VAR
	pTargetData : POINTER TO TcVnRotatedRectangle;
END_VAR
IF NOT IsEquivalentTo(Target) THEN
	RETURN;
END_IF

pTargetData := Target.Address;
activeData REF= pTargetData^;
SetMemberReference();
TryMakeReferenceTo := TRUE;
END_METHOD

PROPERTY PUBLIC Value : REFERENCE TO TcVnRotatedRectangle
GET
Value REF= activeData;
END_GET
END_PROPERTY

PROPERTY PUBLIC aCenter : REFERENCE TO _TcVnPoint2_REAL
GET
aCenter REF= _aCenter;
END_GET
END_PROPERTY

PROPERTY PUBLIC fAngle : REFERENCE TO _REAL
GET
fAngle REF= _fAngle;
END_GET
END_PROPERTY

PROPERTY PUBLIC stSize : REFERENCE TO _TcVnSize2_REAL
GET
stSize REF= _stSize;
END_GET
END_PROPERTY

END_FUNCTION_BLOCK

// Datatypes/Structs/_TcVnSize2_REAL
{attribute 'linkalways'} 
{attribute 'no_explicit_call' := 'This FB is a CLASS and must be accessed using methods or properties'}
{attribute 'enable_dynamic_creation'}
FUNCTION_BLOCK _TcVnSize2_REAL EXTENDS StructuredDatatypeBase
VAR
	localData : TcVnSize2_REAL;
	activeData : REFERENCE TO TcVnSize2_REAL REF= localData;
    _fWidth : _REAL(localdata.fWidth);
    _fHeight : _REAL(localdata.fHeight);
END_VAR

PROPERTY PUBLIC Address : PVOID
GET
Address := ADR(activeData);
END_GET
END_PROPERTY

METHOD PUBLIC ClearReference
VAR_INPUT
END_VAR
activeData REF= localData;
SetMemberReference();
END_METHOD

PROPERTY PUBLIC Size : UDINT
GET
Size := SIZEOF(activeData);
END_GET
END_PROPERTY

METHOD FB_init : BOOL
VAR_INPUT
	bInitRetains : BOOL; // if TRUE, the retain variables are initialized (warm start / cold start)
	bInCopyCode : BOOL;  // if TRUE, the instance afterwards gets moved into the copy code (online change)
END_VAR
SetMemberReference();
AddMember('fWidth', _fWidth);
AddMember('fHeight', _fHeight);
END_METHOD

METHOD PROTECTED SetMemberReference
VAR_INPUT
END_VAR
_fWidth.MakeReferenceTo(activeData.fWidth);
_fHeight.MakeReferenceTo(activeData.fHeight);
END_METHOD

METHOD PUBLIC Clone : I_Datatype
VAR
    pClone : POINTER TO _TcVnSize2_REAL;
END_VAR
pClone := __NEW(_TcVnSize2_REAL());
pClone^.Value := Value;
Clone := pClone^;
END_METHOD

PROPERTY PUBLIC Identifier : T_MAXSTRING
GET
Identifier := 'TcVnSize2_REAL';
END_GET
END_PROPERTY

METHOD PUBLIC MakeReferenceTo
VAR_INPUT
	ReferenceTarget : REFERENCE TO TcVnSize2_REAL;
END_VAR
activeData REF= ReferenceTarget;
SetMemberReference();
END_METHOD

METHOD TryMakeReferenceTo : BOOL
VAR_INPUT
	Target : I_Datatype;
END_VAR
VAR
	pTargetData : POINTER TO TcVnSize2_REAL;
END_VAR
IF NOT IsEquivalentTo(Target) THEN
	RETURN;
END_IF

pTargetData := Target.Address;
activeData REF= pTargetData^;
SetMemberReference();
TryMakeReferenceTo := TRUE;
END_METHOD

PROPERTY PUBLIC Value : REFERENCE TO TcVnSize2_REAL
GET
Value REF= activeData;
END_GET
END_PROPERTY

PROPERTY PUBLIC fHeight : REFERENCE TO _REAL
GET
fHeight REF= _fHeight;
END_GET
END_PROPERTY

PROPERTY PUBLIC fWidth : REFERENCE TO _REAL
GET
fWidth REF= _fWidth;
END_GET
END_PROPERTY

END_FUNCTION_BLOCK

// Datatypes/VisionDatatypePack
{attribute 'linkalways'} 
{attribute 'no_explicit_call' := 'This FB is a CLASS and must be accessed using methods or properties'}
{attribute 'enable_dynamic_creation'}
FUNCTION_BLOCK VisionDatatypePack IMPLEMENTS I_DatatypePack
VAR
    // aliases
    _gVCP_REGISTER_ADDRESS : _GVCP_REGISTER_ADDRESS;
    _tcVnPoint : _TcVnPoint;
    _tcVnPoint2_DINT : _TcVnPoint2_DINT;
    _tcVnPoint2_LREAL : _TcVnPoint2_LREAL;
    _tcVnPoint2_REAL : _TcVnPoint2_REAL;
    _tcVnPoint3_LREAL : _TcVnPoint3_LREAL;
    _tcVnPoint3_REAL : _TcVnPoint3_REAL;
    _tcVnRectangle : _TcVnRectangle;
  
    _tcVnArray10_ITcVnImage : _TcVnArray10_ITcVnImage;
    _tcVnArray3_Point2_REAL : _TcVnArray3_Point2_REAL;
    //_tcVnArray33_UDINT : _TcVnArray33_UDINT;
    _tcVnArray4_LREAL : _TcVnArray4_LREAL;
    _tcVnArray4_Point2_REAL : _TcVnArray4_Point2_REAL;
    _tcVnArray7_LREAL : _TcVnArray7_LREAL;
    _tcVnArray8_LREAL : _TcVnArray8_LREAL;
//    _tcVnMatrix2x3_LREAL : _TcVnMatrix2x3_LREAL;
//    _tcVnMatrix3x3_LREAL : _TcVnMatrix3x3_LREAL;
    _tcVnVector2_DINT : _TcVnVector2_DINT;
    _tcVnVector2_INT : _TcVnVector2_INT;
    _tcVnVector2_LREAL : _TcVnVector2_LREAL;
    _tcVnVector2_REAL : _TcVnVector2_REAL;
    _tcVnVector2_SINT : _TcVnVector2_SINT;
    _tcVnVector2_UINT : _TcVnVector2_UINT;
    _tcVnVector2_USINT : _TcVnVector2_USINT;
    _tcVnVector3_INT : _TcVnVector3_INT;
    _tcVnVector3_LREAL : _TcVnVector3_LREAL;
    _tcVnVector3_REAL : _TcVnVector3_REAL;
    _tcVnVector3_SINT : _TcVnVector3_SINT;
    _tcVnVector3_UINT : _TcVnVector3_UINT;
    _tcVnVector3_USINT : _TcVnVector3_USINT;
    _tcVnVector4_DINT : _TcVnVector4_DINT;
    _tcVnVector4_INT : _TcVnVector4_INT;
    _tcVnVector4_LREAL : _TcVnVector4_LREAL;
    _tcVnVector4_SINT : _TcVnVector4_SINT;
    _tcVnVector4_UINT : _TcVnVector4_UINT;
    _tcVnVector4_USINT : _TcVnVector4_USINT;
 
    // constants
    
    // arrays
    _array0to1OfDINT : _Array0to1OfDINT;
    _array0to1OfINT : _Array0to1OfINT;
    _array0to1OfLREAL : _Array0to1OfLREAL;
    _array0to1OfREAL : _Array0to1OfREAL;
    _array0to1OfSINT : _Array0to1OfSINT;
    _array0to1OfUINT : _Array0to1OfUINT;
    _array0to1OfUSINT : _Array0to1OfUSINT;
    _array0to2OfINT : _Array0to2OfINT;
    _array0to2OfLREAL : _Array0to2OfLREAL;
    _array0to2OfREAL : _Array0to2OfREAL;
    _array0to2OfSINT : _Array0to2OfSINT;
    _array0to2OfUINT : _Array0to2OfUINT;
    _array0to2OfUSINT : _Array0to2OfUSINT;
    _array0to3OfDINT : _Array0to3OfDINT;
    _array0to3OfINT : _Array0to3OfINT;
	_array0to3OfLREAL : _Array0to3OfLREAL;
    _array0to6OfLREAL : _Array0to6OfLREAL;
    _array0to7OfLREAL : _Array0to7OfLREAL;
	_array0to1_0to2OfLREAL : _Array0to1_0to2OfLREAL;
	_array0to2_0to2OfLREAL : _Array0to2_0to2OfLREAL;
    
    // enums
	_eTcVn2dCodeSearchStrategy : _ETcVn2dCodeSearchStrategy(ETcVn2dCodeSearchStrategy.TCVN_CSS_DEFAULT);
	
    // structs
//   _gVSP_IMAGE_INFO : _GVSP_IMAGE_INFO;
//   _gVSP_LEADER_PAYLOAD_IMAGE : _GVSP_LEADER_PAYLOAD_IMAGE;
//  _gVSP_PIXEL_FORMAT : _GVSP_PIXEL_FORMAT;
//  _tcVnCameraCalibrationOptions : _TcVnCameraCalibrationOptions;
    _tcVnCircularArc : _TcVnCircularArc;
//  _tcVnCodeGrades1D : _TcVnCodeGrades1D;
//  _tcVnCodeGradesDM : _TcVnCodeGradesDM;
//  _tcVnCodeGradesQR : _TcVnCodeGradesQR;
    _tcVnDMatch : _TcVnDMatch;
	_tcVnImageInfo : _TcVnImageInfo;
    _tcVnKeyPoint : _TcVnKeyPoint;
//  _tcVnMatrix : _TcVnMatrix;
//  _tcVnMoments : _TcVnMoments;
//  _tcVnParamsAGAST : _TcVnParamsAGAST;
//  _tcVnParamsAKAZE : _TcVnParamsAKAZE;
    _tcVnParamsBlobDetection : _TcVnParamsBlobDetection;
//  _tcVnParamsBRISK : _TcVnParamsBRISK;
//  _tcVnParamsFAST : _TcVnParamsFAST;
//  _tcVnParamsGFTT : _TcVnParamsGFTT;
//  _tcVnParamsKAZE : _TcVnParamsKAZE;
//  _tcVnParamsMSER : _TcVnParamsMSER;
//  _tcVnParamsORB : _TcVnParamsORB;
//  _tcVnParamsSB : _TcVnParamsSB;
    _tcVnPixelFormat : _TcVnPixelFormat;
	_tcVnRectangle_DINT : _TcVnRectangle_DINT;
    _tcVnRectangle_UDINT : _TcVnRectangle_UDINT;
    _tcVnRotatedRectangle : _TcVnRotatedRectangle;
    _tcVnSize2_REAL : _TcVnSize2_REAL;
	
	// interfaces
	_iTcVnImage : _ITcVnImage;
	
END_VAR

METHOD RegisterWithDatatypes
VAR_INPUT
	Datatypes : I_Datatypes;
END_VAR
// aliases
Datatypes.RegisterDatatype(_GVCP_REGISTER_ADDRESS);
Datatypes.RegisterDatatype(_tcVnPoint);
Datatypes.RegisterDatatype(_tcVnPoint2_DINT);
Datatypes.RegisterDatatype(_tcVnPoint2_LREAL);
Datatypes.RegisterDatatype(_tcVnPoint2_REAL);
Datatypes.RegisterDatatype(_tcVnPoint3_LREAL);
Datatypes.RegisterDatatype(_tcVnPoint3_REAL);
Datatypes.RegisterDatatype(_tcVnRectangle);

Datatypes.RegisterDatatype(_tcVnArray10_ITcVnImage);
Datatypes.RegisterDatatype(_tcVnArray3_Point2_REAL);
//Datatypes.RegisterDatatype(_tcVnArray33_UDINT);
Datatypes.RegisterDatatype(_tcVnArray4_LREAL);
Datatypes.RegisterDatatype(_tcVnArray4_Point2_REAL);
Datatypes.RegisterDatatype(_tcVnArray7_LREAL);
Datatypes.RegisterDatatype(_tcVnArray8_LREAL);
//Datatypes.RegisterDatatype(_tcVnMatrix2x3_LREAL);
//Datatypes.RegisterDatatype(_tcVnMatrix3x3_LREAL);
Datatypes.RegisterDatatype(_tcVnVector2_DINT);
Datatypes.RegisterDatatype(_tcVnVector2_INT);
Datatypes.RegisterDatatype(_tcVnVector2_LREAL);
Datatypes.RegisterDatatype(_tcVnVector2_REAL);
Datatypes.RegisterDatatype(_tcVnVector2_SINT);
Datatypes.RegisterDatatype(_tcVnVector2_UINT);
Datatypes.RegisterDatatype(_tcVnVector2_USINT);
Datatypes.RegisterDatatype(_tcVnVector3_INT);
Datatypes.RegisterDatatype(_tcVnVector3_LREAL);
Datatypes.RegisterDatatype(_tcVnVector3_REAL);
Datatypes.RegisterDatatype(_tcVnVector3_SINT);
Datatypes.RegisterDatatype(_tcVnVector3_UINT);
Datatypes.RegisterDatatype(_tcVnVector3_USINT);
Datatypes.RegisterDatatype(_tcVnVector4_DINT);
Datatypes.RegisterDatatype(_tcVnVector4_INT);
Datatypes.RegisterDatatype(_tcVnVector4_LREAL);
Datatypes.RegisterDatatype(_tcVnVector4_SINT);
Datatypes.RegisterDatatype(_tcVnVector4_UINT);
Datatypes.RegisterDatatype(_tcVnVector4_USINT);

// constants

// arrays
Datatypes.RegisterDatatype(_array0to1OfDINT);
Datatypes.RegisterDatatype(_array0to1OfINT);
Datatypes.RegisterDatatype(_array0to1OfLREAL);
Datatypes.RegisterDatatype(_array0to1OfREAL);
Datatypes.RegisterDatatype(_array0to1OfSINT);
Datatypes.RegisterDatatype(_array0to1OfUINT);
Datatypes.RegisterDatatype(_array0to1OfUSINT);
Datatypes.RegisterDatatype(_array0to2OfINT);
Datatypes.RegisterDatatype(_array0to2OfLREAL);
Datatypes.RegisterDatatype(_array0to2OfREAL);
Datatypes.RegisterDatatype(_array0to2OfSINT);
Datatypes.RegisterDatatype(_array0to2OfUINT);
Datatypes.RegisterDatatype(_array0to2OfUSINT);
Datatypes.RegisterDatatype(_array0to3OfDINT);
Datatypes.RegisterDatatype(_array0to3OfINT);
Datatypes.RegisterDatatype(_array0to3OfLREAL);
Datatypes.RegisterDatatype(_array0to6OfLREAL);
Datatypes.RegisterDatatype(_array0to7OfLREAL);
Datatypes.RegisterDatatype(_array0to1_0to2OfLREAL);
Datatypes.RegisterDatatype(_array0to2_0to2OfLREAL);

// enums
Datatypes.RegisterDatatype(_eTcVn2dCodeSearchStrategy);

// structs
//Datatypes.RegisterDatatype(_gVSP_IMAGE_INFO);
//Datatypes.RegisterDatatype(_gVSP_LEADER_PAYLOAD_IMAGE);
//Datatypes.RegisterDatatype(_gVSP_PIXEL_FORMAT);
//Datatypes.RegisterDatatype(_tcVnCameraCalibrationOptions);
Datatypes.RegisterDatatype(_tcVnCircularArc);
//Datatypes.RegisterDatatype(_tcVnCodeGrades1D);
//Datatypes.RegisterDatatype(_tcVnCodeGradesDM);
//Datatypes.RegisterDatatype(_tcVnCodeGradesQR);
Datatypes.RegisterDatatype(_tcVnDMatch);
Datatypes.RegisterDatatype(_tcVnImageInfo);
Datatypes.RegisterDatatype(_tcVnKeyPoint);
//Datatypes.RegisterDatatype(_tcVnMatrix);
//Datatypes.RegisterDatatype(_tcVnMoments);
//Datatypes.RegisterDatatype(_tcVnParamsAGAST);
//Datatypes.RegisterDatatype(_tcVnParamsAKAZE);
Datatypes.RegisterDatatype(_tcVnParamsBlobDetection);
//Datatypes.RegisterDatatype(_tcVnParamsBRISK);
//Datatypes.RegisterDatatype(_tcVnParamsFAST);
//Datatypes.RegisterDatatype(_tcVnParamsGFTT);
//Datatypes.RegisterDatatype(_tcVnParamsKAZE);
//Datatypes.RegisterDatatype(_tcVnParamsMSER);
//Datatypes.RegisterDatatype(_tcVnParamsORB);
//Datatypes.RegisterDatatype(_tcVnParamsSB);
Datatypes.RegisterDatatype(_tcVnPixelFormat);
Datatypes.RegisterDatatype(_tcVnRectangle_DINT);
Datatypes.RegisterDatatype(_tcVnRectangle_UDINT);
Datatypes.RegisterDatatype(_tcVnRotatedRectangle);
Datatypes.RegisterDatatype(_tcVnSize2_REAL);

// interfaces
Datatypes.RegisterDatatype(_iTcVnImage);
END_METHOD

END_FUNCTION_BLOCK

// Nodes/Algebraic Image Operations/Node_F_VN_BitwiseAndImages
{attribute 'linkalways'} 
{attribute 'no_explicit_call' := 'This FB is a CLASS and must be accessed using methods or properties'}
{attribute 'enable_dynamic_creation'}
FUNCTION_BLOCK Node_F_VN_BitwiseAndImages EXTENDS VisionNode
VAR
    ipSrcImage1 : _ITcVnImage;
    ipSrcImage2 : _ITcVnImage;
    ipDestImage : _ITcVnImage;
    hrPrev : _HRESULT(S_OK);
	hresult : _HRESULT(S_OK);
END_VAR

METHOD FB_init : BOOL
VAR_INPUT
	bInitRetains : BOOL; // if TRUE, the retain variables are initialized (warm start / cold start)
	bInCopyCode : BOOL;  // if TRUE, the instance afterwards gets moved into the copy code (online change)
END_VAR
AddInput('ipSrcImage1', ipSrcImage1);
AddInput('ipSrcImage2', ipSrcImage2);
AddInput('hrPrev', hrPrev);
AddOutput('ipDestImage', ipDestImage);
AddOutput('hresult',hresult);
END_METHOD

METHOD PUBLIC  Clone : I_Node
VAR
	pNode : POINTER TO Node_F_VN_BitwiseAndImages;
END_VAR
pNode := __NEW(Node_F_VN_BitwiseAndImages);
Clone := pNode^;
END_METHOD

METHOD PROTECTED OnExecute : HRESULT
hresult.Value := F_VN_BitwiseAndImages(
    ipSrcImage1 := ipSrcImage1.Value,
    ipSrcImage2 := ipSrcImage2.Value,
	ipDestImage := ipDestImage.Value,
	hrPrev:= hrPrev.Value);
END_METHOD

METHOD PUBLIC PreExecutionCheck
VAR_INPUT
	Check : I_PreExecutionChecks;
END_VAR
Check.IsTrue(ipSrcImage1.IsValid, 'ipSrcImage1 must contain an image');
Check.IsTrue(ipSrcImage2.IsValid, 'ipSrcImage2 must contain an image');
END_METHOD

END_FUNCTION_BLOCK

// Nodes/VisionNode/VisionNode
FUNCTION_BLOCK ABSTRACT VisionNode EXTENDS Node IMPLEMENTS I_PreCheckedNode
VAR
	preExecutionCheckExtension : PreExecutionCheckExtension('precheck', THIS^);
END_VAR

METHOD PUBLIC ABSTRACT PreExecutionCheck
VAR_INPUT
	Check : I_PreExecutionChecks;
END_VAR
END_METHOD

END_FUNCTION_BLOCK

// Nodes/Algebraic Image Operations/Node_F_VN_BitwiseNotImage
{attribute 'linkalways'} 
{attribute 'no_explicit_call' := 'This FB is a CLASS and must be accessed using methods or properties'}
{attribute 'enable_dynamic_creation'}
FUNCTION_BLOCK Node_F_VN_BitwiseNotImage EXTENDS VisionNode
VAR
    ipSrcImage : _ITcVnImage;
    ipDestImage : _ITcVnImage;
    hrPrev : _HRESULT(S_OK);
	hresult : _HRESULT(S_OK);
END_VAR

METHOD FB_init : BOOL
VAR_INPUT
	bInitRetains : BOOL; // if TRUE, the retain variables are initialized (warm start / cold start)
	bInCopyCode : BOOL;  // if TRUE, the instance afterwards gets moved into the copy code (online change)
END_VAR
AddInput('ipSrcImage', ipSrcImage);
AddInput('hrPrev', hrPrev);
AddOutput('ipDestImage', ipDestImage);
AddOutput('hresult',hresult);
END_METHOD

METHOD PUBLIC  Clone : I_Node
VAR
	pNode : POINTER TO Node_F_VN_BitwiseNotImage;
END_VAR
pNode := __NEW(Node_F_VN_BitwiseNotImage);
Clone := pNode^;
END_METHOD

METHOD PROTECTED OnExecute : HRESULT
hresult.Value := F_VN_BitwiseNotImage(
    ipSrcImage := ipSrcImage.Value,
	ipDestImage := ipDestImage.Value,
	hrPrev:= hrPrev.Value);
END_METHOD

METHOD PUBLIC PreExecutionCheck
VAR_INPUT
	Check : I_PreExecutionChecks;
END_VAR
Check.IsTrue(ipSrcImage.IsValid, 'ipSrcImage must contain an image');
END_METHOD

END_FUNCTION_BLOCK

// Nodes/Algebraic Image Operations/Node_F_VN_BitwiseOrImages
{attribute 'linkalways'} 
{attribute 'no_explicit_call' := 'This FB is a CLASS and must be accessed using methods or properties'}
{attribute 'enable_dynamic_creation'}
FUNCTION_BLOCK Node_F_VN_BitwiseOrImages EXTENDS VisionNode
VAR
    ipSrcImage1 : _ITcVnImage;
    ipSrcImage2 : _ITcVnImage;
    ipDestImage : _ITcVnImage;
    hrPrev : _HRESULT(S_OK);
	hresult : _HRESULT(S_OK);
END_VAR

METHOD FB_init : BOOL
VAR_INPUT
	bInitRetains : BOOL; // if TRUE, the retain variables are initialized (warm start / cold start)
	bInCopyCode : BOOL;  // if TRUE, the instance afterwards gets moved into the copy code (online change)
END_VAR
AddInput('ipSrcImage1', ipSrcImage1);
AddInput('ipSrcImage2', ipSrcImage2);
AddInput('hrPrev', hrPrev);
AddOutput('ipDestImage', ipDestImage);
AddOutput('hresult',hresult);
END_METHOD

METHOD PUBLIC  Clone : I_Node
VAR
	pNode : POINTER TO Node_F_VN_BitwiseOrImages;
END_VAR
pNode := __NEW(Node_F_VN_BitwiseOrImages);
Clone := pNode^;
END_METHOD

METHOD PROTECTED OnExecute : HRESULT
hresult.Value := F_VN_BitwiseOrImages(
    ipSrcImage1 := ipSrcImage1.Value,
    ipSrcImage2 := ipSrcImage2.Value,
	ipDestImage := ipDestImage.Value,
	hrPrev:= hrPrev.Value);
END_METHOD

METHOD PUBLIC PreExecutionCheck
VAR_INPUT
	Check : I_PreExecutionChecks;
END_VAR
Check.IsTrue(ipSrcImage1.IsValid, 'ipSrcImage1 must contain an image');
Check.IsTrue(ipSrcImage2.IsValid, 'ipSrcImage2 must contain an image');
END_METHOD

END_FUNCTION_BLOCK

// Nodes/Algebraic Image Operations/Node_F_VN_BitwiseXorImages
{attribute 'linkalways'} 
{attribute 'no_explicit_call' := 'This FB is a CLASS and must be accessed using methods or properties'}
{attribute 'enable_dynamic_creation'}
FUNCTION_BLOCK Node_F_VN_BitwiseXorImages EXTENDS VisionNode
VAR
    ipSrcImage1 : _ITcVnImage;
    ipSrcImage2 : _ITcVnImage;
    ipDestImage : _ITcVnImage;
    hrPrev : _HRESULT(S_OK);
	hresult : _HRESULT(S_OK);
END_VAR

METHOD FB_init : BOOL
VAR_INPUT
	bInitRetains : BOOL; // if TRUE, the retain variables are initialized (warm start / cold start)
	bInCopyCode : BOOL;  // if TRUE, the instance afterwards gets moved into the copy code (online change)
END_VAR
AddInput('ipSrcImage1', ipSrcImage1);
AddInput('ipSrcImage2', ipSrcImage2);
AddInput('hrPrev', hrPrev);
AddOutput('ipDestImage', ipDestImage);
AddOutput('hresult',hresult);
END_METHOD

METHOD PUBLIC  Clone : I_Node
VAR
	pNode : POINTER TO Node_F_VN_BitwiseXorImages;
END_VAR
pNode := __NEW(Node_F_VN_BitwiseXorImages);
Clone := pNode^;
END_METHOD

METHOD PROTECTED OnExecute : HRESULT
hresult.Value := F_VN_BitwiseXorImages(
    ipSrcImage1 := ipSrcImage1.Value,
    ipSrcImage2 := ipSrcImage2.Value,
	ipDestImage := ipDestImage.Value,
	hrPrev:= hrPrev.Value);
END_METHOD

METHOD PUBLIC PreExecutionCheck
VAR_INPUT
	Check : I_PreExecutionChecks;
END_VAR
Check.IsTrue(ipSrcImage1.IsValid, 'ipSrcImage1 must contain an image');
Check.IsTrue(ipSrcImage2.IsValid, 'ipSrcImage2 must contain an image');
END_METHOD

END_FUNCTION_BLOCK

// Nodes/Basic Container Operations/Node_F_VN_AppendToContainer_DINT
{attribute 'linkalways'} 
{attribute 'no_explicit_call' := 'This FB is a CLASS and must be accessed using methods or properties'}
{attribute 'enable_dynamic_creation'}
FUNCTION_BLOCK Node_F_VN_AppendToContainer_DINT EXTENDS VisionNode
VAR
    nElement : _DINT(0);
    ipContainer : _ITcVnContainer;
    hrPrev : _HRESULT(S_OK);
	hresult : _HRESULT(S_OK);
END_VAR

METHOD FB_init : BOOL
VAR_INPUT
	bInitRetains : BOOL; // if TRUE, the retain variables are initialized (warm start / cold start)
	bInCopyCode : BOOL;  // if TRUE, the instance afterwards gets moved into the copy code (online change)
END_VAR
AddInput('nElement', nElement);
AddInput('ipContainer', ipContainer);
AddInput('hrPrev', hrPrev);
AddOutput('ipContainer', ipContainer);
AddOutput('hresult',hresult);
END_METHOD

METHOD PUBLIC  Clone : I_Node
VAR
	pNode : POINTER TO Node_F_VN_AppendToContainer_DINT;
END_VAR
pNode := __NEW(Node_F_VN_AppendToContainer_DINT);
Clone := pNode^;
END_METHOD

METHOD PROTECTED OnExecute : HRESULT
hresult.Value := F_VN_AppendToContainer_DINT(
    nElement := nElement.Value,
	ipContainer := ipContainer.Value,
	hrPrev:= hrPrev.Value);
END_METHOD

METHOD PUBLIC PreExecutionCheck
VAR_INPUT
	Check : I_PreExecutionChecks;
END_VAR
Check.IsTrue(ipContainer.IsValid, 'ipContainer must be a valid container');
Check.IsTrue(ipContainer.HasType('CTcVnContainer_Vector_DINT'), 'ipContainer contains incorrect types');
END_METHOD

END_FUNCTION_BLOCK

// Nodes/Basic Container Operations/Node_F_VN_AppendToContainer_INT
{attribute 'linkalways'} 
{attribute 'no_explicit_call' := 'This FB is a CLASS and must be accessed using methods or properties'}
{attribute 'enable_dynamic_creation'}
FUNCTION_BLOCK Node_F_VN_AppendToContainer_INT EXTENDS VisionNode
VAR
    nElement : _INT(0);
    ipContainer : _ITcVnContainer;
    hrPrev : _HRESULT(S_OK);
	hresult : _HRESULT(S_OK);
END_VAR

METHOD FB_init : BOOL
VAR_INPUT
	bInitRetains : BOOL; // if TRUE, the retain variables are initialized (warm start / cold start)
	bInCopyCode : BOOL;  // if TRUE, the instance afterwards gets moved into the copy code (online change)
END_VAR
AddInput('nElement', nElement);
AddInput('ipContainer', ipContainer);
AddInput('hrPrev', hrPrev);
AddOutput('ipContainer', ipContainer);
AddOutput('hresult',hresult);
END_METHOD

METHOD PUBLIC  Clone : I_Node
VAR
	pNode : POINTER TO Node_F_VN_AppendToContainer_INT;
END_VAR
pNode := __NEW(Node_F_VN_AppendToContainer_INT);
Clone := pNode^;
END_METHOD

METHOD PROTECTED OnExecute : HRESULT
hresult.Value := F_VN_AppendToContainer_INT(
    nElement := nElement.Value,
	ipContainer := ipContainer.Value,
	hrPrev:= hrPrev.Value);
END_METHOD

METHOD PUBLIC PreExecutionCheck
VAR_INPUT
	Check : I_PreExecutionChecks;
END_VAR
Check.IsTrue(ipContainer.IsValid, 'ipContainer must be a valid container');
Check.IsTrue(ipContainer.HasType('CTcVnContainer_Vector_INT'), 'ipContainer contains incorrect types');
END_METHOD

END_FUNCTION_BLOCK

// Nodes/Basic Container Operations/Node_F_VN_AppendToContainer_ITcVnContainer
{attribute 'linkalways'} 
{attribute 'no_explicit_call' := 'This FB is a CLASS and must be accessed using methods or properties'}
{attribute 'enable_dynamic_creation'}
FUNCTION_BLOCK Node_F_VN_AppendToContainer_ITcVnContainer EXTENDS VisionNode
VAR
    ipElement : _ITcVnContainer;
    ipContainer : _ITcVnContainer;
    hrPrev : _HRESULT(S_OK);
	hresult : _HRESULT(S_OK);
END_VAR

METHOD FB_init : BOOL
VAR_INPUT
	bInitRetains : BOOL; // if TRUE, the retain variables are initialized (warm start / cold start)
	bInCopyCode : BOOL;  // if TRUE, the instance afterwards gets moved into the copy code (online change)
END_VAR
AddInput('ipElement', ipElement);
AddInput('ipContainer', ipContainer);
AddInput('hrPrev', hrPrev);
AddOutput('ipContainer', ipContainer);
AddOutput('hresult',hresult);
END_METHOD

METHOD PUBLIC  Clone : I_Node
VAR
	pNode : POINTER TO Node_F_VN_AppendToContainer_ITcVnContainer;
END_VAR
pNode := __NEW(Node_F_VN_AppendToContainer_ITcVnContainer);
Clone := pNode^;
END_METHOD

METHOD PROTECTED OnExecute : HRESULT
hresult.Value := F_VN_AppendToContainer_ITcVnContainer(
    ipElement := ipElement.Value,
	ipContainer := ipContainer.Value,
	hrPrev:= hrPrev.Value);
END_METHOD

METHOD PUBLIC PreExecutionCheck
VAR_INPUT
	Check : I_PreExecutionChecks;
END_VAR
Check.IsTrue(ipContainer.IsValid, 'ipContainer must be a valid container');
END_METHOD

END_FUNCTION_BLOCK

